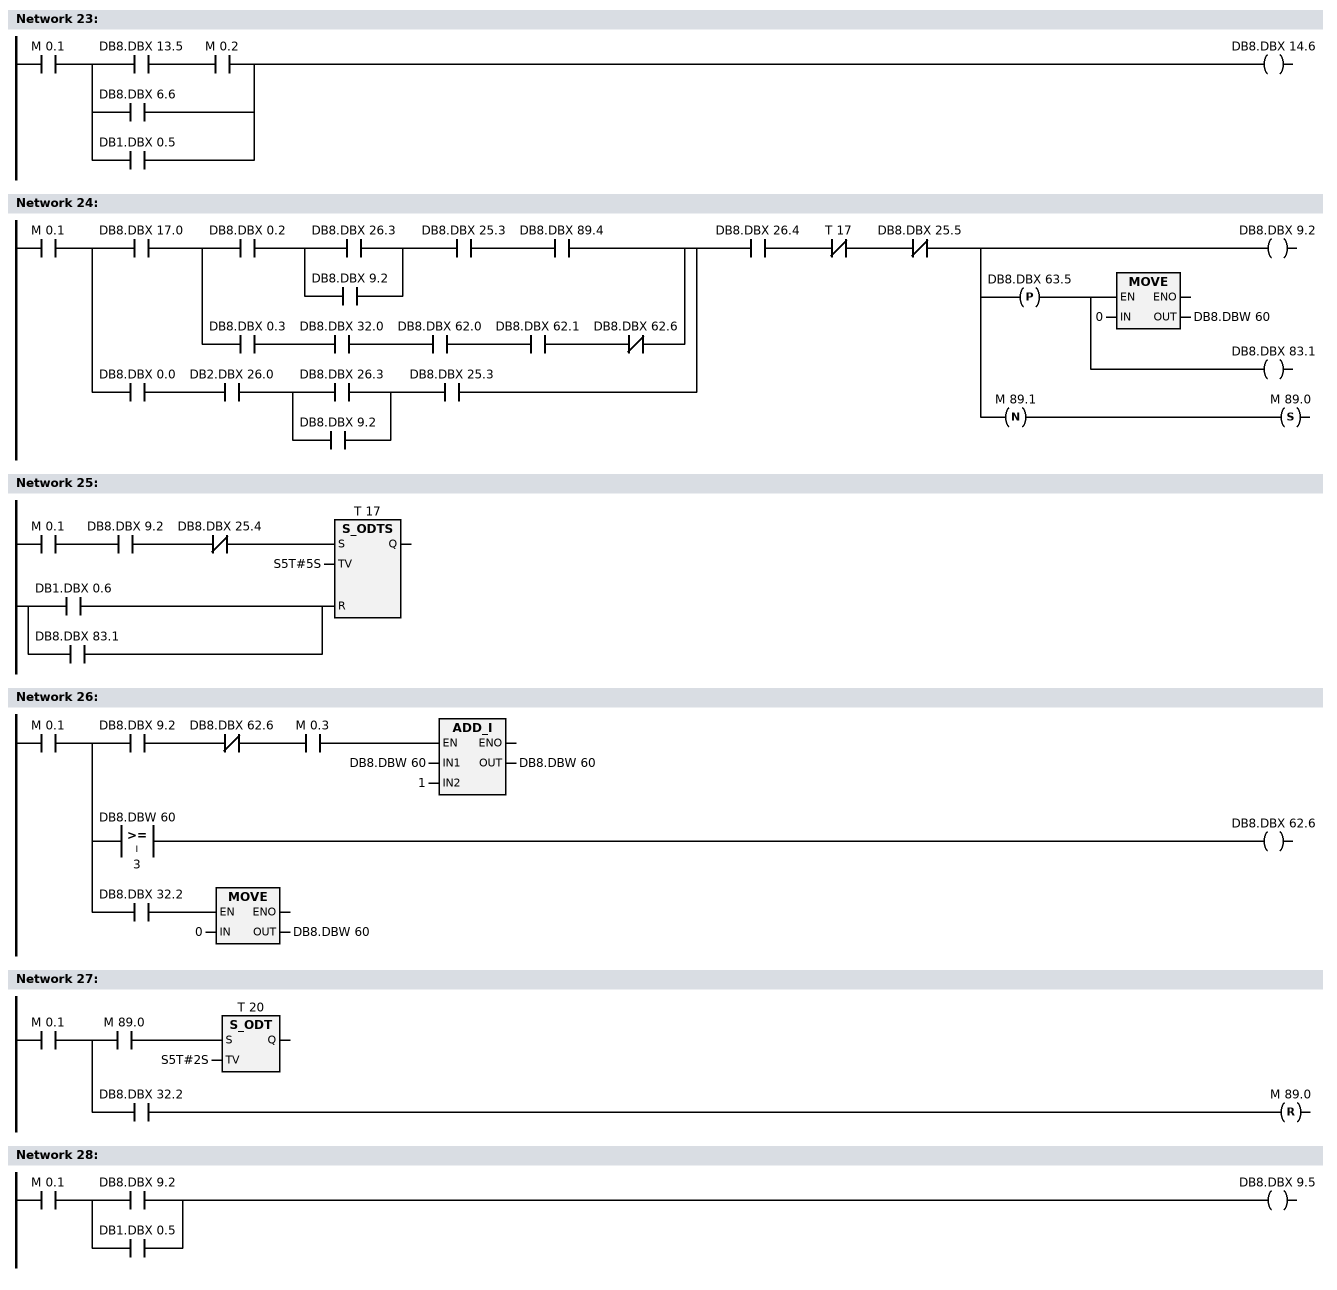
NETWORK
TITLE =
      A     M 0.1;
      A(;
      A     DB8.DBX 13.5;
      A     M 0.2;
      O     DB8.DBX 6.6;
      O     DB1.DBX 0.5;
      );
      =     DB8.DBX 14.6;
NETWORK
TITLE =
      A     M 0.1;
      A(;
      A     DB8.DBX 17.0;
      A(;
      A     DB8.DBX 0.2;
      A(;
      O     DB8.DBX 26.3;
      O     DB8.DBX 9.2;
      );
      A     DB8.DBX 25.3;
      A     DB8.DBX 89.4;
      O;
      A     DB8.DBX 0.3;
      A     DB8.DBX 32.0;
      A     DB8.DBX 62.0;
      A     DB8.DBX 62.1;
      AN    DB8.DBX 62.6;
      );
      O;
      A     DB8.DBX 0.0;
      A     DB2.DBX 26.0;
      A(;
      O     DB8.DBX 26.3;
      O     DB8.DBX 9.2;
      );
      A     DB8.DBX 25.3;
      );
      A     DB8.DBX 26.4;
      AN    T 17;
      AN    DB8.DBX 25.5;
      =     L 0.0;
      A     L 0.0;
      BLD   102;
      =     DB8.DBX 9.2;
      A     L 0.0;
      FP    DB8.DBX 63.5;
      =     L 0.1;
      A     L 0.1;
      JNB   M012;
      L     0;
      T     DB8.DBW 60;
M012: NOP   0;
      A     L 0.1;
      BLD   102;
      =     DB8.DBX 83.1;
      A     L 0.0;
      FN    M 89.1;
      S     M 89.0;
NETWORK
TITLE =
      A     M 0.1;
      A     DB8.DBX 9.2;
      AN    DB8.DBX 25.4;
      L     S5T#5S;
      SS    T 17;
      A(;
      O     DB1.DBX 0.6;
      O     DB8.DBX 83.1;
      );
      R     T 17;
      NOP   0;
      NOP   0;
      NOP   0;
NETWORK
TITLE =
      A     M 0.1;
      =     L 0.0;
      A     L 0.0;
      A     DB8.DBX 9.2;
      AN    DB8.DBX 62.6;
      A     M 0.3;
      JNB   M013;
      L     DB8.DBW 60;
      L     1;
      +I;
      T     DB8.DBW 60;
M013: NOP   0;
      A     L 0.0;
      A(;
      L     DB8.DBW 60;
      L     3;
      >=I;
      );
      =     DB8.DBX 62.6;
      A     L 0.0;
      A     DB8.DBX 32.2;
      JNB   M014;
      L     0;
      T     DB8.DBW 60;
M014: NOP   0;
NETWORK
TITLE =
      A     M 0.1;
      =     L 0.0;
      A     L 0.0;
      A     M 89.0;
      L     S5T#2S;
      SD    T 20;
      NOP   0;
      NOP   0;
      NOP   0;
      NOP   0;
      A     L 0.0;
      A     DB8.DBX 32.2;
      R     M 89.0;
NETWORK
TITLE =
      A     M 0.1;
      A(;
      O     DB8.DBX 9.2;
      O     DB1.DBX 0.5;
      );
      =     DB8.DBX 9.5;
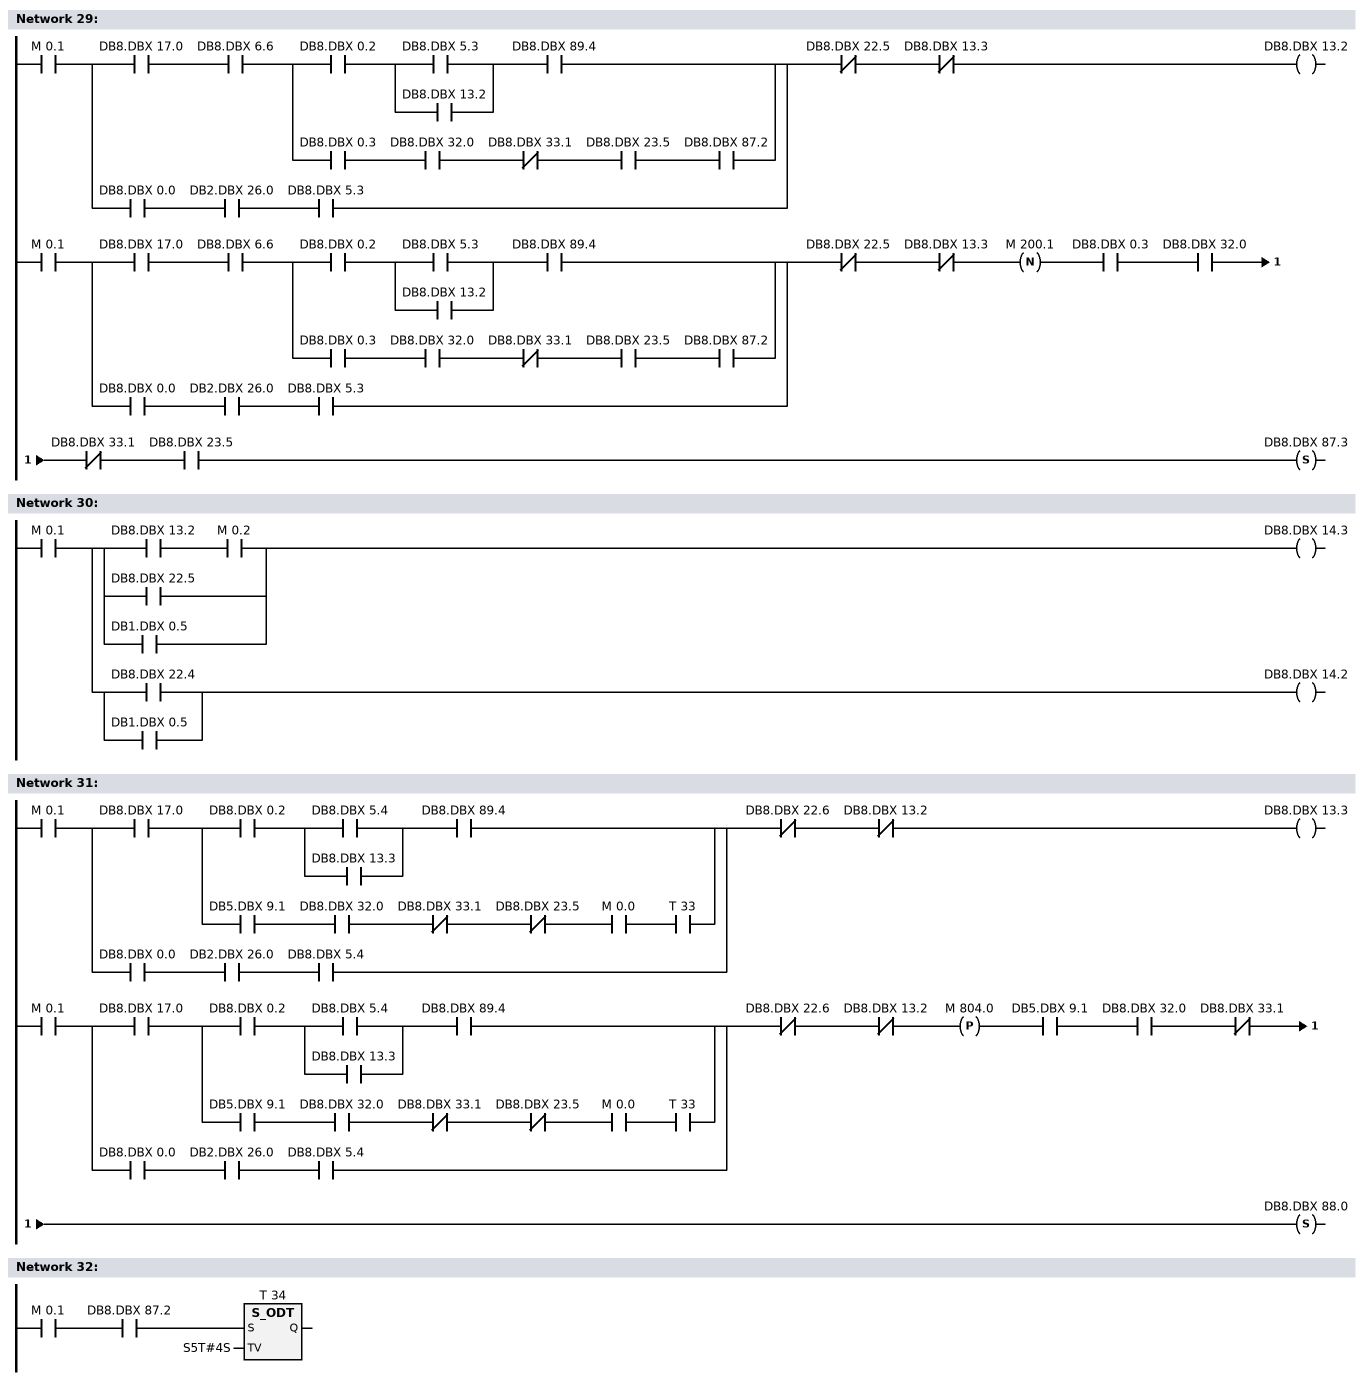
NETWORK
TITLE =
      A     M 0.1;
      A(;
      A     DB8.DBX 17.0;
      A     DB8.DBX 6.6;
      A(;
      A     DB8.DBX 0.2;
      A(;
      O     DB8.DBX 5.3;
      O     DB8.DBX 13.2;
      );
      A     DB8.DBX 89.4;
      O;
      A     DB8.DBX 0.3;
      A     DB8.DBX 32.0;
      AN    DB8.DBX 33.1;
      A     DB8.DBX 23.5;
      A     DB8.DBX 87.2;
      );
      O;
      A     DB8.DBX 0.0;
      A     DB2.DBX 26.0;
      A     DB8.DBX 5.3;
      );
      AN    DB8.DBX 22.5;
      AN    DB8.DBX 13.3;
      =     L 0.0;
      A     L 0.0;
      BLD   102;
      =     DB8.DBX 13.2;
      A(;
      A     L 0.0;
      FN    M 200.1;
      );
      A     DB8.DBX 0.3;
      A     DB8.DBX 32.0;
      AN    DB8.DBX 33.1;
      A     DB8.DBX 23.5;
      S     DB8.DBX 87.3;
NETWORK
TITLE =
      A     M 0.1;
      =     L 0.0;
      A     L 0.0;
      A(;
      A     DB8.DBX 13.2;
      A     M 0.2;
      O     DB8.DBX 22.5;
      O     DB1.DBX 0.5;
      );
      =     DB8.DBX 14.3;
      A     L 0.0;
      A(;
      O     DB8.DBX 22.4;
      O     DB1.DBX 0.5;
      );
      =     DB8.DBX 14.2;
NETWORK
TITLE =
      A     M 0.1;
      A(;
      A     DB8.DBX 17.0;
      A(;
      A     DB8.DBX 0.2;
      A(;
      O     DB8.DBX 5.4;
      O     DB8.DBX 13.3;
      );
      A     DB8.DBX 89.4;
      O;
      A     DB5.DBX 9.1;
      A     DB8.DBX 32.0;
      AN    DB8.DBX 33.1;
      AN    DB8.DBX 23.5;
      A     M 0.0;
      A     T 33;
      );
      O;
      A     DB8.DBX 0.0;
      A     DB2.DBX 26.0;
      A     DB8.DBX 5.4;
      );
      AN    DB8.DBX 22.6;
      AN    DB8.DBX 13.2;
      =     L 0.0;
      A     L 0.0;
      BLD   102;
      =     DB8.DBX 13.3;
      A(;
      A     L 0.0;
      FP    M 804.0;
      );
      A     DB5.DBX 9.1;
      A     DB8.DBX 32.0;
      AN    DB8.DBX 33.1;
      S     DB8.DBX 88.0;
NETWORK
TITLE =
      A     M 0.1;
      A     DB8.DBX 87.2;
      L     S5T#4S;
      SD    T 34;
      NOP   0;
      NOP   0;
      NOP   0;
      NOP   0;
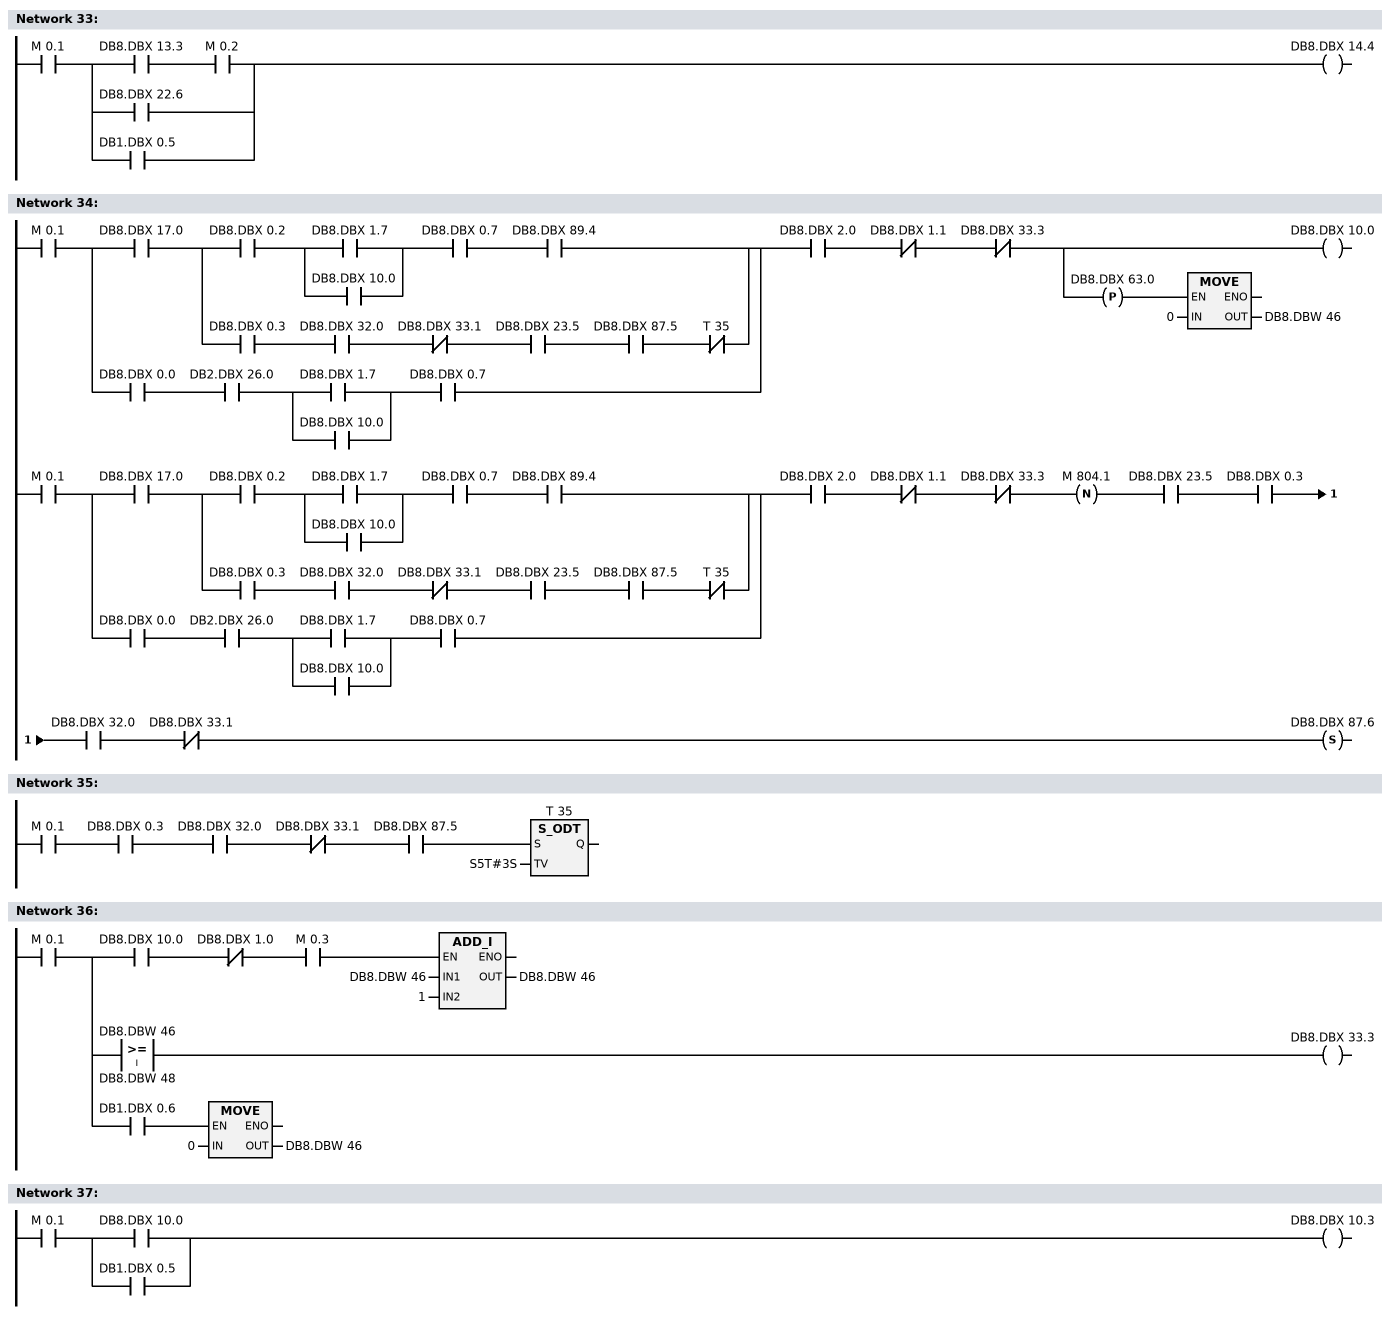
NETWORK
TITLE =
      A     M 0.1;
      A(;
      A     DB8.DBX 13.3;
      A     M 0.2;
      O     DB8.DBX 22.6;
      O     DB1.DBX 0.5;
      );
      =     DB8.DBX 14.4;
NETWORK
TITLE =
      A     M 0.1;
      A(;
      A     DB8.DBX 17.0;
      A(;
      A     DB8.DBX 0.2;
      A(;
      O     DB8.DBX 1.7;
      O     DB8.DBX 10.0;
      );
      A     DB8.DBX 0.7;
      A     DB8.DBX 89.4;
      O;
      A     DB8.DBX 0.3;
      A     DB8.DBX 32.0;
      AN    DB8.DBX 33.1;
      A     DB8.DBX 23.5;
      A     DB8.DBX 87.5;
      AN    T 35;
      );
      O;
      A     DB8.DBX 0.0;
      A     DB2.DBX 26.0;
      A(;
      O     DB8.DBX 1.7;
      O     DB8.DBX 10.0;
      );
      A     DB8.DBX 0.7;
      );
      A     DB8.DBX 2.0;
      AN    DB8.DBX 1.1;
      AN    DB8.DBX 33.3;
      =     L 0.0;
      A     L 0.0;
      BLD   102;
      =     DB8.DBX 10.0;
      A     L 0.0;
      FP    DB8.DBX 63.0;
      JNB   M015;
      L     0;
      T     DB8.DBW 46;
M015: NOP   0;
      A(;
      A     L 0.0;
      FN    M 804.1;
      );
      A     DB8.DBX 23.5;
      A     DB8.DBX 0.3;
      A     DB8.DBX 32.0;
      AN    DB8.DBX 33.1;
      S     DB8.DBX 87.6;
NETWORK
TITLE =
      A     M 0.1;
      A     DB8.DBX 0.3;
      A     DB8.DBX 32.0;
      AN    DB8.DBX 33.1;
      A     DB8.DBX 87.5;
      L     S5T#3S;
      SD    T 35;
      NOP   0;
      NOP   0;
      NOP   0;
      NOP   0;
NETWORK
TITLE =
      A     M 0.1;
      =     L 0.0;
      A     L 0.0;
      A     DB8.DBX 10.0;
      AN    DB8.DBX 1.0;
      A     M 0.3;
      JNB   M016;
      L     DB8.DBW 46;
      L     1;
      +I;
      T     DB8.DBW 46;
M016: NOP   0;
      A     L 0.0;
      A(;
      L     DB8.DBW 46;
      L     DB8.DBW 48;
      >=I;
      );
      =     DB8.DBX 33.3;
      A     L 0.0;
      A     DB1.DBX 0.6;
      JNB   M017;
      L     0;
      T     DB8.DBW 46;
M017: NOP   0;
NETWORK
TITLE =
      A     M 0.1;
      A(;
      O     DB8.DBX 10.0;
      O     DB1.DBX 0.5;
      );
      =     DB8.DBX 10.3;
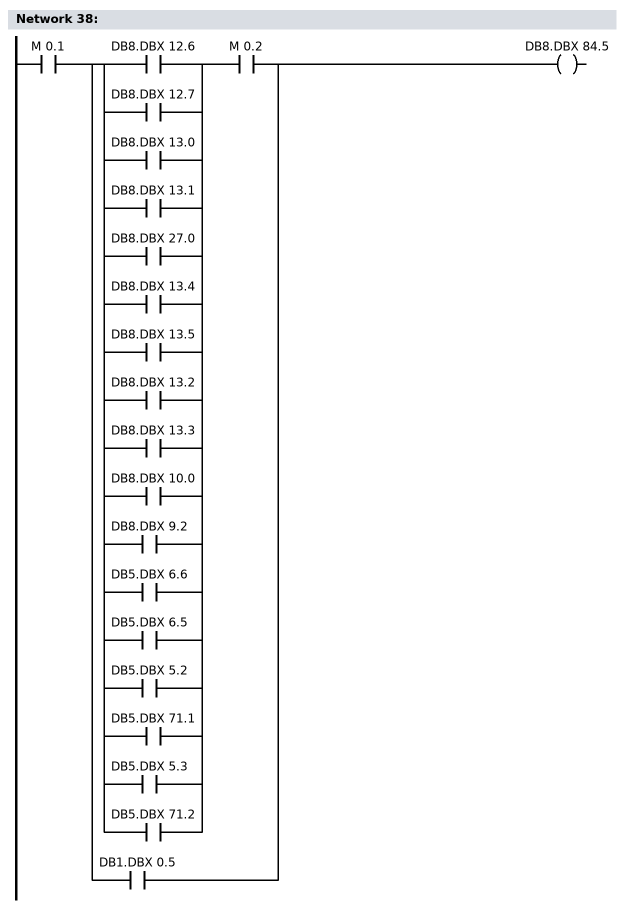
NETWORK
TITLE =
      A     M 0.1;
      A(;
      A(;
      O     DB8.DBX 12.6;
      O     DB8.DBX 12.7;
      O     DB8.DBX 13.0;
      O     DB8.DBX 13.1;
      O     DB8.DBX 27.0;
      O     DB8.DBX 13.4;
      O     DB8.DBX 13.5;
      O     DB8.DBX 13.2;
      O     DB8.DBX 13.3;
      O     DB8.DBX 10.0;
      O     DB8.DBX 9.2;
      O     DB5.DBX 6.6;
      O     DB5.DBX 6.5;
      O     DB5.DBX 5.2;
      O     DB5.DBX 71.1;
      O     DB5.DBX 5.3;
      O     DB5.DBX 71.2;
      );
      A     M 0.2;
      O     DB1.DBX 0.5;
      );
      =     DB8.DBX 84.5;
END_FUNCTION

FUNCTION FC 14 : VOID
AUTHOR : Arun
VERSION : 0.1
BEGIN
// (block stored without names or comments; labels and parameter names are numbered)
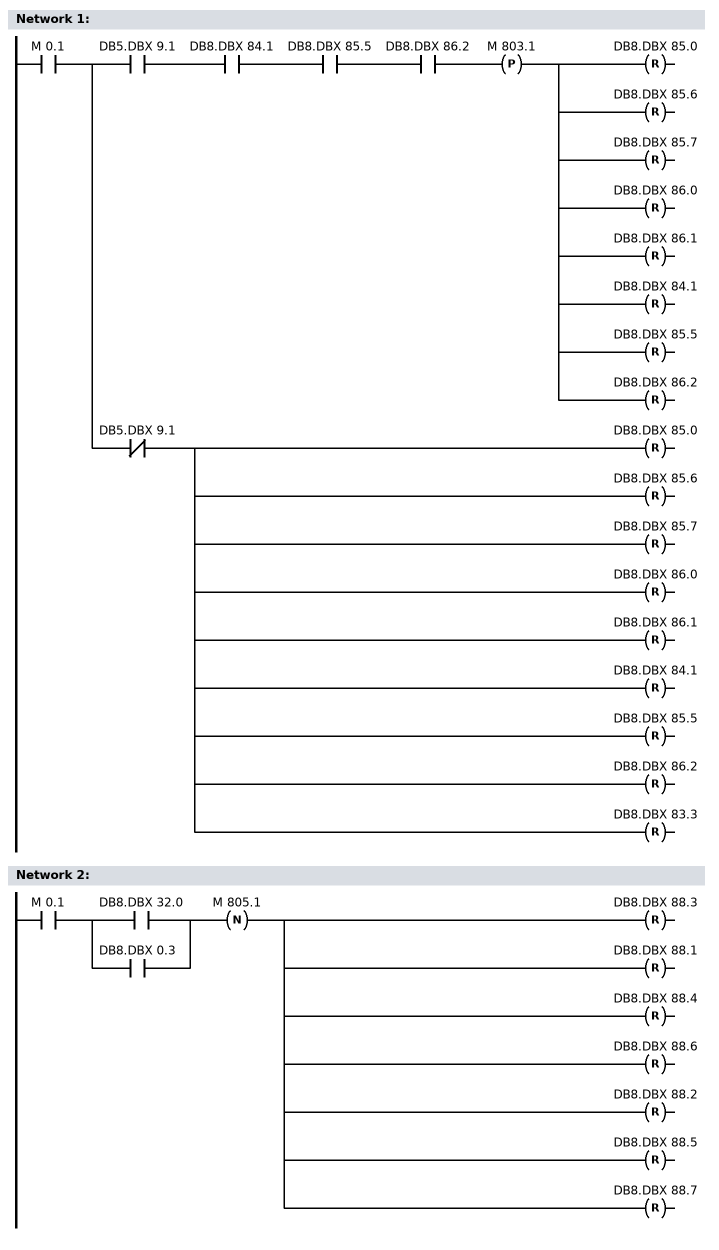
NETWORK
TITLE =
      A     M 0.1;
      =     L 0.0;
      A     L 0.0;
      A     DB5.DBX 9.1;
      A     DB8.DBX 84.1;
      A     DB8.DBX 85.5;
      A     DB8.DBX 86.2;
      FP    M 803.1;
      R     DB8.DBX 85.0;
      R     DB8.DBX 85.6;
      R     DB8.DBX 85.7;
      R     DB8.DBX 86.0;
      R     DB8.DBX 86.1;
      R     DB8.DBX 84.1;
      R     DB8.DBX 85.5;
      R     DB8.DBX 86.2;
      A     L 0.0;
      AN    DB5.DBX 9.1;
      R     DB8.DBX 85.0;
      R     DB8.DBX 85.6;
      R     DB8.DBX 85.7;
      R     DB8.DBX 86.0;
      R     DB8.DBX 86.1;
      R     DB8.DBX 84.1;
      R     DB8.DBX 85.5;
      R     DB8.DBX 86.2;
      R     DB8.DBX 83.3;
NETWORK
TITLE =
      A     M 0.1;
      A(;
      O     DB8.DBX 32.0;
      O     DB8.DBX 0.3;
      );
      FN    M 805.1;
      R     DB8.DBX 88.3;
      R     DB8.DBX 88.1;
      R     DB8.DBX 88.4;
      R     DB8.DBX 88.6;
      R     DB8.DBX 88.2;
      R     DB8.DBX 88.5;
      R     DB8.DBX 88.7;
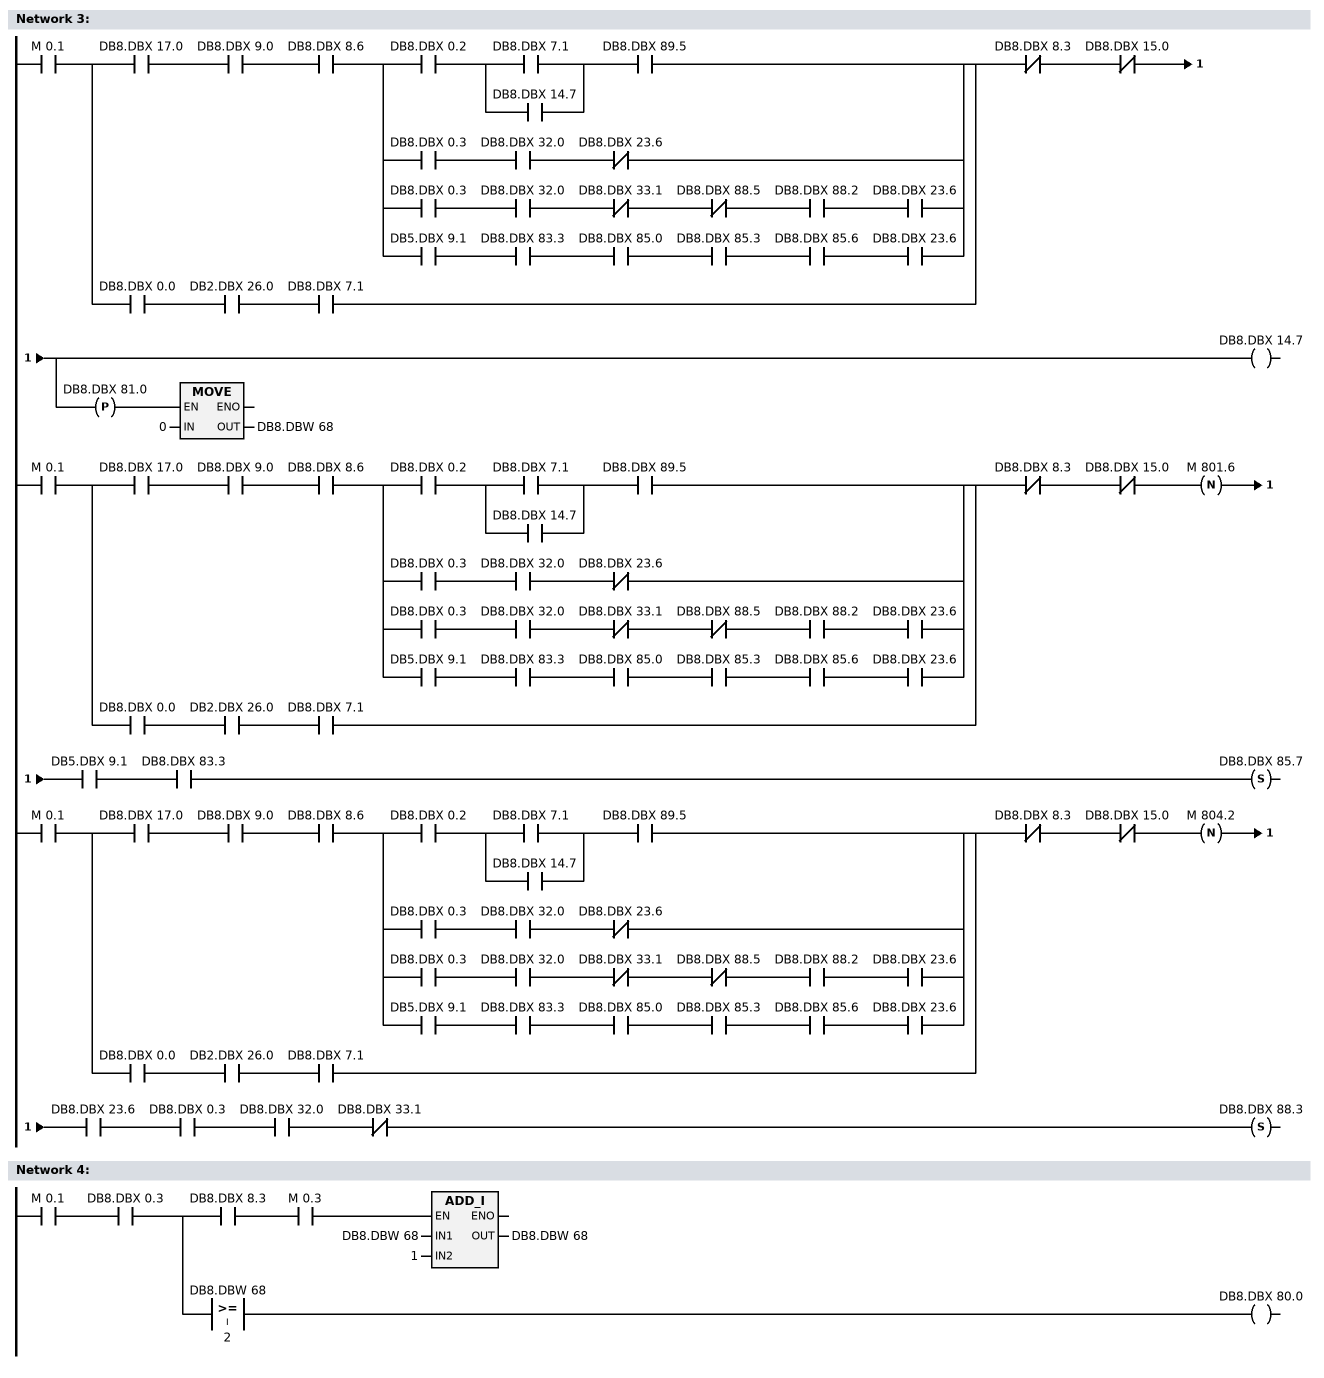
NETWORK
TITLE =
      A     M 0.1;
      A(;
      A     DB8.DBX 17.0;
      A     DB8.DBX 9.0;
      A     DB8.DBX 8.6;
      A(;
      A     DB8.DBX 0.2;
      A(;
      O     DB8.DBX 7.1;
      O     DB8.DBX 14.7;
      );
      A     DB8.DBX 89.5;
      O;
      A     DB8.DBX 0.3;
      A     DB8.DBX 32.0;
      AN    DB8.DBX 23.6;
      O;
      A     DB8.DBX 0.3;
      A     DB8.DBX 32.0;
      AN    DB8.DBX 33.1;
      AN    DB8.DBX 88.5;
      A     DB8.DBX 88.2;
      A     DB8.DBX 23.6;
      O;
      A     DB5.DBX 9.1;
      A     DB8.DBX 83.3;
      A     DB8.DBX 85.0;
      A     DB8.DBX 85.3;
      A     DB8.DBX 85.6;
      A     DB8.DBX 23.6;
      );
      O;
      A     DB8.DBX 0.0;
      A     DB2.DBX 26.0;
      A     DB8.DBX 7.1;
      );
      AN    DB8.DBX 8.3;
      AN    DB8.DBX 15.0;
      =     L 0.0;
      A     L 0.0;
      BLD   102;
      =     DB8.DBX 14.7;
      A     L 0.0;
      FP    DB8.DBX 81.0;
      JNB   M001;
      L     0;
      T     DB8.DBW 68;
M001: NOP   0;
      A(;
      A     L 0.0;
      FN    M 801.6;
      );
      A     DB5.DBX 9.1;
      A     DB8.DBX 83.3;
      S     DB8.DBX 85.7;
      A(;
      A     L 0.0;
      FN    M 804.2;
      );
      A     DB8.DBX 23.6;
      A     DB8.DBX 0.3;
      A     DB8.DBX 32.0;
      AN    DB8.DBX 33.1;
      S     DB8.DBX 88.3;
NETWORK
TITLE =
      A     M 0.1;
      A     DB8.DBX 0.3;
      =     L 0.0;
      A     L 0.0;
      A     DB8.DBX 8.3;
      A     M 0.3;
      JNB   M002;
      L     DB8.DBW 68;
      L     1;
      +I;
      T     DB8.DBW 68;
M002: NOP   0;
      A     L 0.0;
      A(;
      L     DB8.DBW 68;
      L     2;
      >=I;
      );
      =     DB8.DBX 80.0;
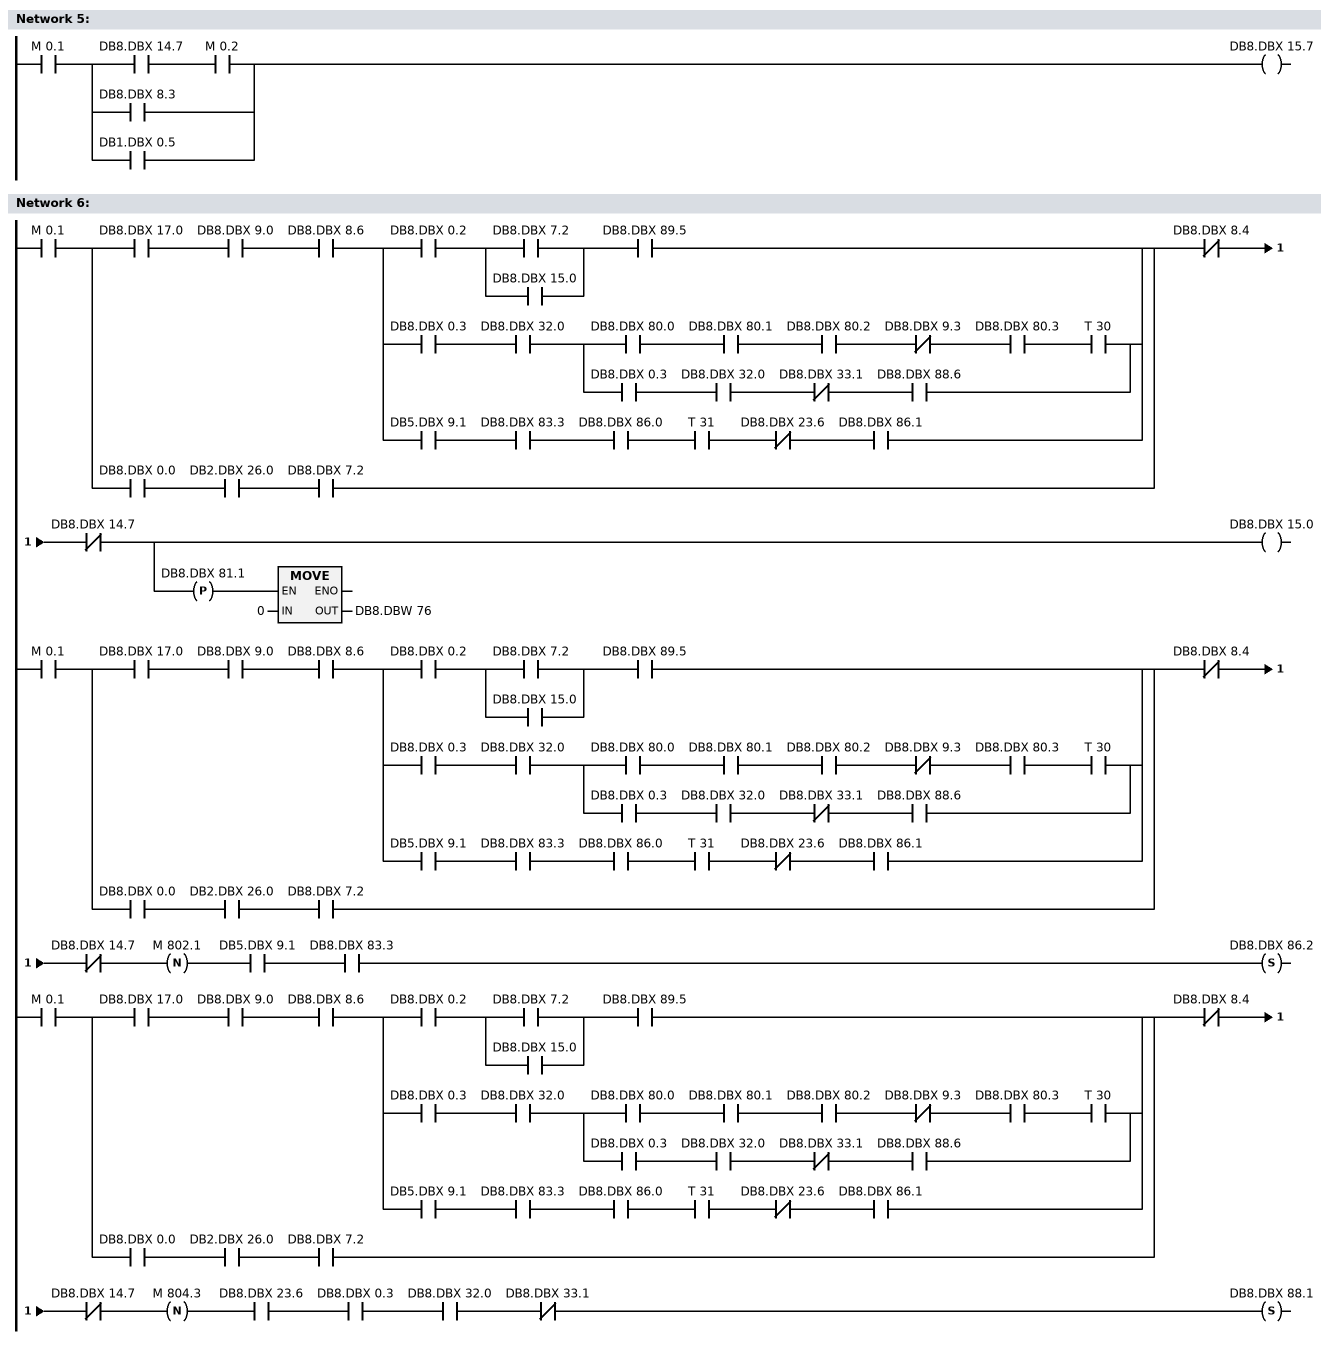
NETWORK
TITLE =
      A     M 0.1;
      A(;
      A     DB8.DBX 14.7;
      A     M 0.2;
      O     DB8.DBX 8.3;
      O     DB1.DBX 0.5;
      );
      =     DB8.DBX 15.7;
NETWORK
TITLE =
      A     M 0.1;
      A(;
      A     DB8.DBX 17.0;
      A     DB8.DBX 9.0;
      A     DB8.DBX 8.6;
      A(;
      A     DB8.DBX 0.2;
      A(;
      O     DB8.DBX 7.2;
      O     DB8.DBX 15.0;
      );
      A     DB8.DBX 89.5;
      O;
      A     DB8.DBX 0.3;
      A     DB8.DBX 32.0;
      A(;
      A     DB8.DBX 80.0;
      A     DB8.DBX 80.1;
      A     DB8.DBX 80.2;
      AN    DB8.DBX 9.3;
      A     DB8.DBX 80.3;
      A     T 30;
      O;
      A     DB8.DBX 0.3;
      A     DB8.DBX 32.0;
      AN    DB8.DBX 33.1;
      A     DB8.DBX 88.6;
      );
      O;
      A     DB5.DBX 9.1;
      A     DB8.DBX 83.3;
      A     DB8.DBX 86.0;
      A     T 31;
      AN    DB8.DBX 23.6;
      A     DB8.DBX 86.1;
      );
      O;
      A     DB8.DBX 0.0;
      A     DB2.DBX 26.0;
      A     DB8.DBX 7.2;
      );
      AN    DB8.DBX 8.4;
      AN    DB8.DBX 14.7;
      =     L 0.0;
      A     L 0.0;
      BLD   102;
      =     DB8.DBX 15.0;
      A     L 0.0;
      FP    DB8.DBX 81.1;
      JNB   M003;
      L     0;
      T     DB8.DBW 76;
M003: NOP   0;
      A(;
      A     L 0.0;
      FN    M 802.1;
      );
      A     DB5.DBX 9.1;
      A     DB8.DBX 83.3;
      S     DB8.DBX 86.2;
      A(;
      A     L 0.0;
      FN    M 804.3;
      );
      A     DB8.DBX 23.6;
      A     DB8.DBX 0.3;
      A     DB8.DBX 32.0;
      AN    DB8.DBX 33.1;
      S     DB8.DBX 88.1;
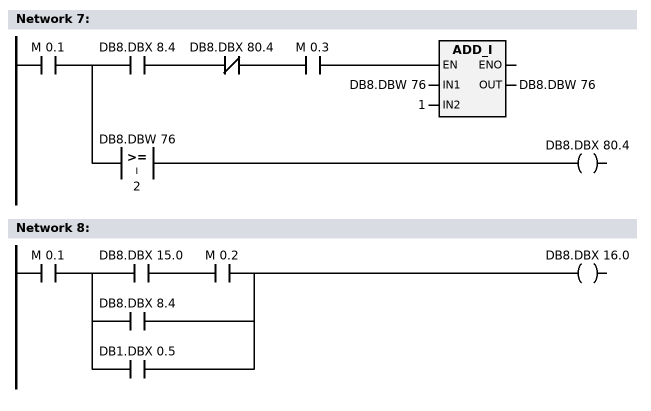
NETWORK
TITLE =
      A     M 0.1;
      =     L 0.0;
      A     L 0.0;
      A     DB8.DBX 8.4;
      AN    DB8.DBX 80.4;
      A     M 0.3;
      JNB   M004;
      L     DB8.DBW 76;
      L     1;
      +I;
      T     DB8.DBW 76;
M004: NOP   0;
      A     L 0.0;
      A(;
      L     DB8.DBW 76;
      L     2;
      >=I;
      );
      =     DB8.DBX 80.4;
NETWORK
TITLE =
      A     M 0.1;
      A(;
      A     DB8.DBX 15.0;
      A     M 0.2;
      O     DB8.DBX 8.4;
      O     DB1.DBX 0.5;
      );
      =     DB8.DBX 16.0;
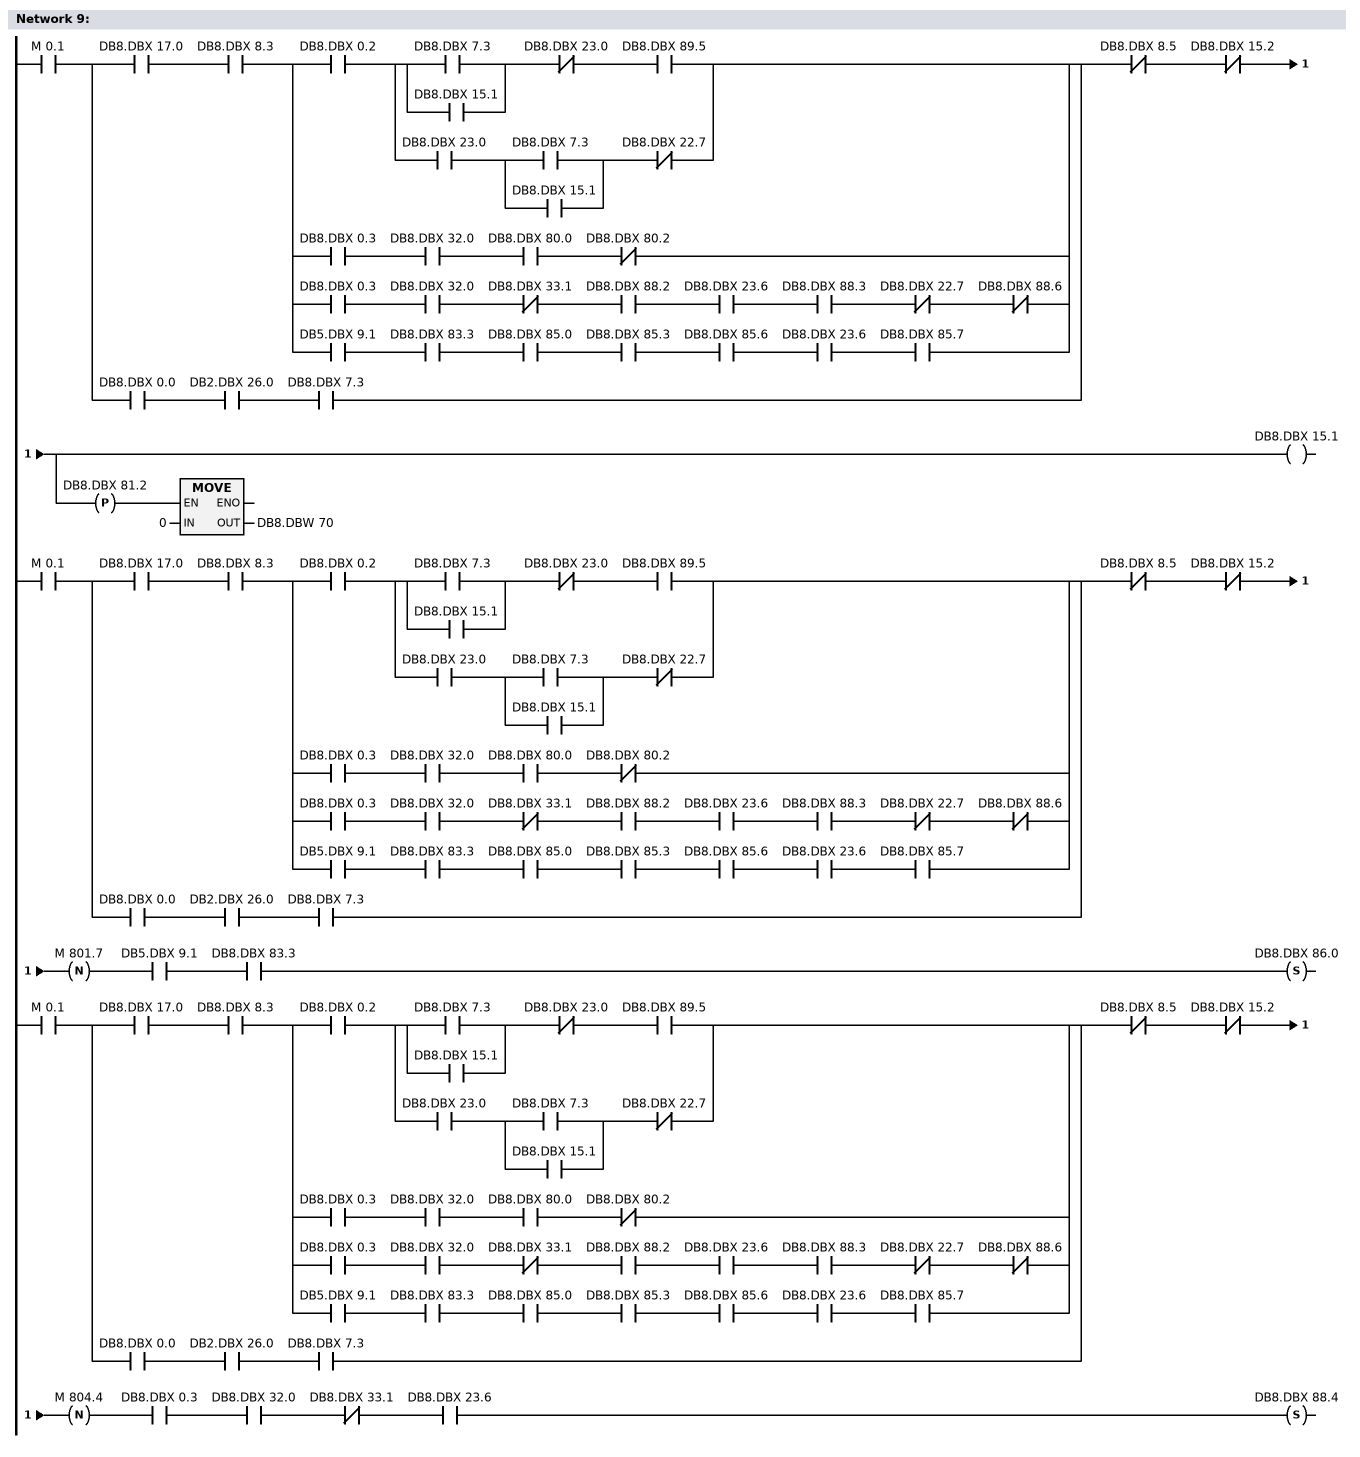
NETWORK
TITLE =
      A     M 0.1;
      A(;
      A     DB8.DBX 17.0;
      A     DB8.DBX 8.3;
      A(;
      A     DB8.DBX 0.2;
      A(;
      A(;
      O     DB8.DBX 7.3;
      O     DB8.DBX 15.1;
      );
      AN    DB8.DBX 23.0;
      A     DB8.DBX 89.5;
      O;
      A     DB8.DBX 23.0;
      A(;
      O     DB8.DBX 7.3;
      O     DB8.DBX 15.1;
      );
      AN    DB8.DBX 22.7;
      );
      O;
      A     DB8.DBX 0.3;
      A     DB8.DBX 32.0;
      A     DB8.DBX 80.0;
      AN    DB8.DBX 80.2;
      O;
      A     DB8.DBX 0.3;
      A     DB8.DBX 32.0;
      AN    DB8.DBX 33.1;
      A     DB8.DBX 88.2;
      A     DB8.DBX 23.6;
      A     DB8.DBX 88.3;
      AN    DB8.DBX 22.7;
      AN    DB8.DBX 88.6;
      O;
      A     DB5.DBX 9.1;
      A     DB8.DBX 83.3;
      A     DB8.DBX 85.0;
      A     DB8.DBX 85.3;
      A     DB8.DBX 85.6;
      A     DB8.DBX 23.6;
      A     DB8.DBX 85.7;
      );
      O;
      A     DB8.DBX 0.0;
      A     DB2.DBX 26.0;
      A     DB8.DBX 7.3;
      );
      AN    DB8.DBX 8.5;
      AN    DB8.DBX 15.2;
      =     L 0.0;
      A     L 0.0;
      BLD   102;
      =     DB8.DBX 15.1;
      A     L 0.0;
      FP    DB8.DBX 81.2;
      JNB   M005;
      L     0;
      T     DB8.DBW 70;
M005: NOP   0;
      A(;
      A     L 0.0;
      FN    M 801.7;
      );
      A     DB5.DBX 9.1;
      A     DB8.DBX 83.3;
      S     DB8.DBX 86.0;
      A(;
      A     L 0.0;
      FN    M 804.4;
      );
      A     DB8.DBX 0.3;
      A     DB8.DBX 32.0;
      AN    DB8.DBX 33.1;
      A     DB8.DBX 23.6;
      S     DB8.DBX 88.4;
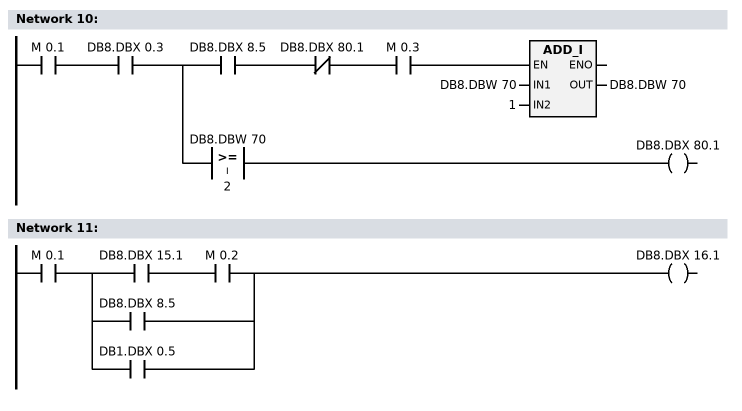
NETWORK
TITLE =
      A     M 0.1;
      A     DB8.DBX 0.3;
      =     L 0.0;
      A     L 0.0;
      A     DB8.DBX 8.5;
      AN    DB8.DBX 80.1;
      A     M 0.3;
      JNB   M006;
      L     DB8.DBW 70;
      L     1;
      +I;
      T     DB8.DBW 70;
M006: NOP   0;
      A     L 0.0;
      A(;
      L     DB8.DBW 70;
      L     2;
      >=I;
      );
      =     DB8.DBX 80.1;
NETWORK
TITLE =
      A     M 0.1;
      A(;
      A     DB8.DBX 15.1;
      A     M 0.2;
      O     DB8.DBX 8.5;
      O     DB1.DBX 0.5;
      );
      =     DB8.DBX 16.1;
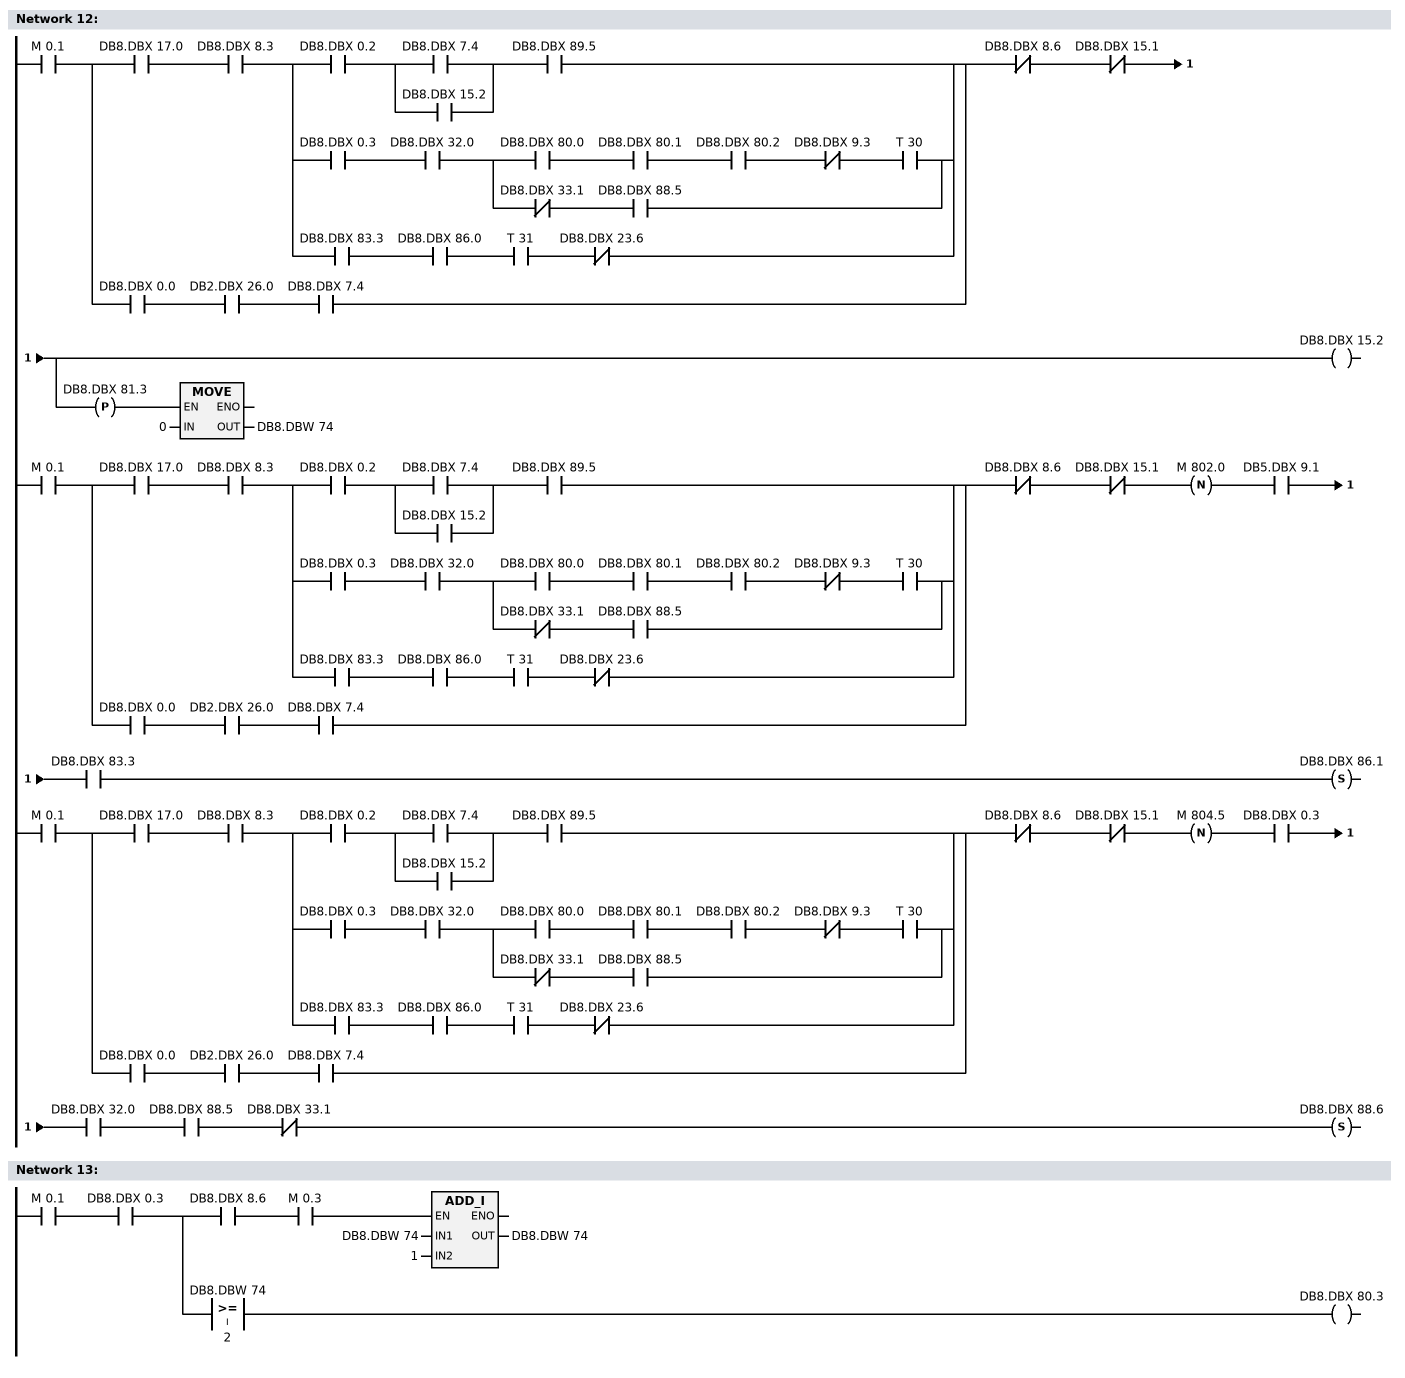
NETWORK
TITLE =
      A     M 0.1;
      A(;
      A     DB8.DBX 17.0;
      A     DB8.DBX 8.3;
      A(;
      A     DB8.DBX 0.2;
      A(;
      O     DB8.DBX 7.4;
      O     DB8.DBX 15.2;
      );
      A     DB8.DBX 89.5;
      O;
      A     DB8.DBX 0.3;
      A     DB8.DBX 32.0;
      A(;
      A     DB8.DBX 80.0;
      A     DB8.DBX 80.1;
      A     DB8.DBX 80.2;
      AN    DB8.DBX 9.3;
      A     T 30;
      O;
      AN    DB8.DBX 33.1;
      A     DB8.DBX 88.5;
      );
      O;
      A     DB8.DBX 83.3;
      A     DB8.DBX 86.0;
      A     T 31;
      AN    DB8.DBX 23.6;
      );
      O;
      A     DB8.DBX 0.0;
      A     DB2.DBX 26.0;
      A     DB8.DBX 7.4;
      );
      AN    DB8.DBX 8.6;
      AN    DB8.DBX 15.1;
      =     L 0.0;
      A     L 0.0;
      BLD   102;
      =     DB8.DBX 15.2;
      A     L 0.0;
      FP    DB8.DBX 81.3;
      JNB   M007;
      L     0;
      T     DB8.DBW 74;
M007: NOP   0;
      A(;
      A     L 0.0;
      FN    M 802.0;
      );
      A     DB5.DBX 9.1;
      A     DB8.DBX 83.3;
      S     DB8.DBX 86.1;
      A(;
      A     L 0.0;
      FN    M 804.5;
      );
      A     DB8.DBX 0.3;
      A     DB8.DBX 32.0;
      A     DB8.DBX 88.5;
      AN    DB8.DBX 33.1;
      S     DB8.DBX 88.6;
NETWORK
TITLE =
      A     M 0.1;
      A     DB8.DBX 0.3;
      =     L 0.0;
      A     L 0.0;
      A     DB8.DBX 8.6;
      A     M 0.3;
      JNB   M008;
      L     DB8.DBW 74;
      L     1;
      +I;
      T     DB8.DBW 74;
M008: NOP   0;
      A     L 0.0;
      A(;
      L     DB8.DBW 74;
      L     2;
      >=I;
      );
      =     DB8.DBX 80.3;
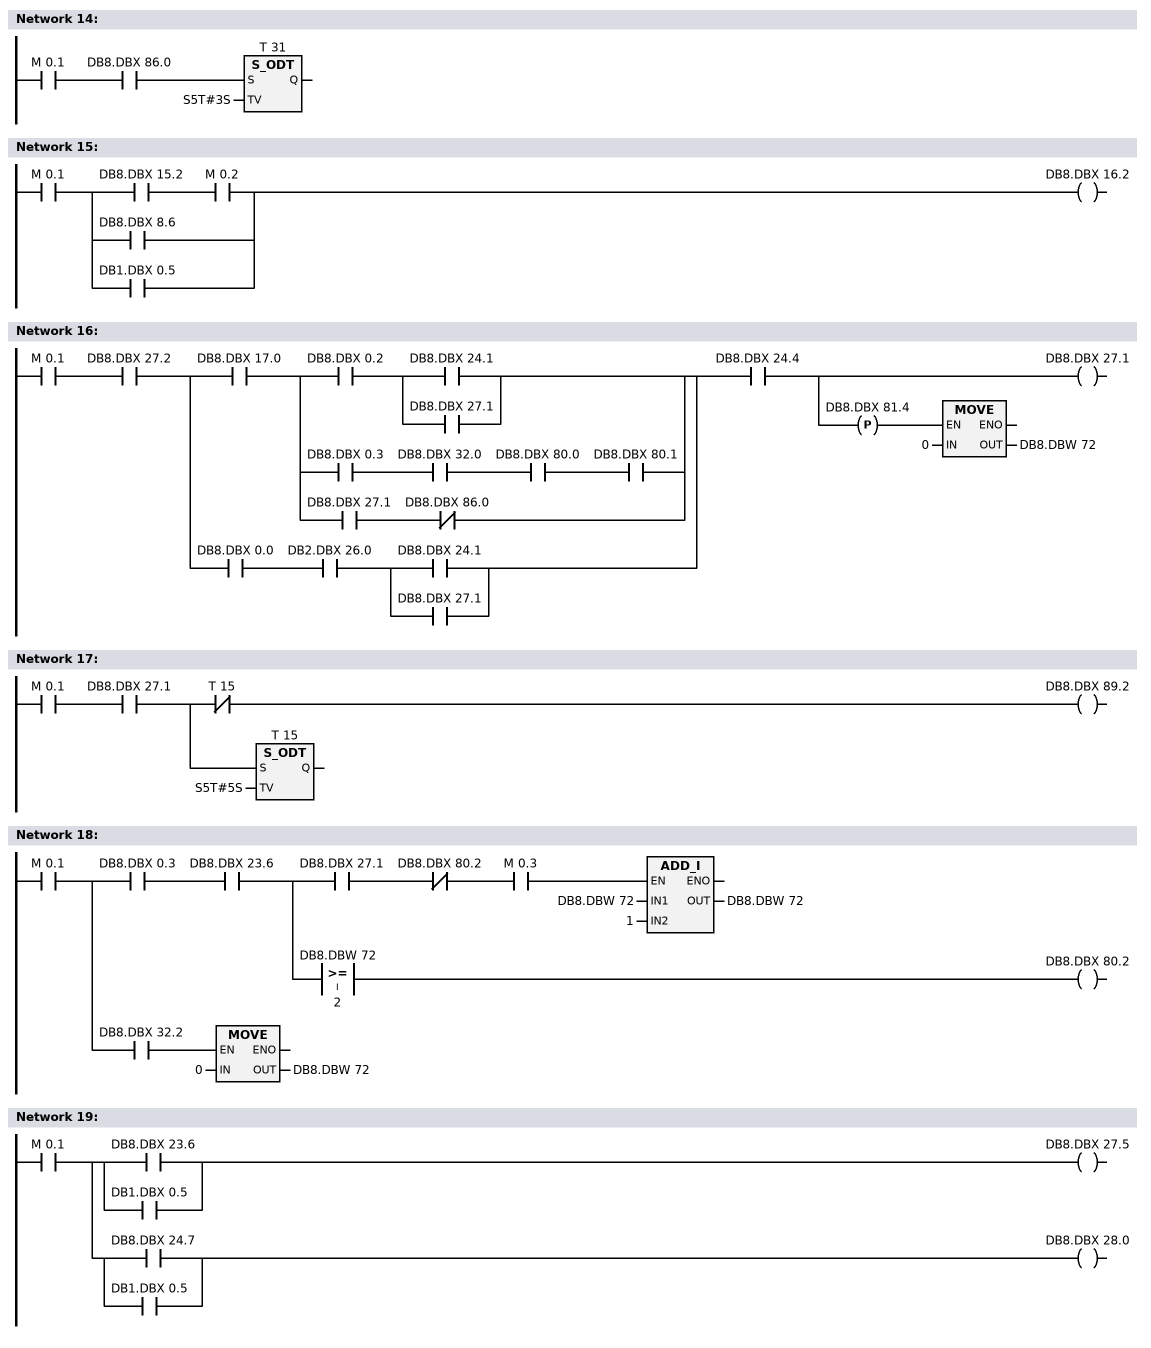
NETWORK
TITLE =
      A     M 0.1;
      A     DB8.DBX 86.0;
      L     S5T#3S;
      SD    T 31;
      NOP   0;
      NOP   0;
      NOP   0;
      NOP   0;
NETWORK
TITLE =
      A     M 0.1;
      A(;
      A     DB8.DBX 15.2;
      A     M 0.2;
      O     DB8.DBX 8.6;
      O     DB1.DBX 0.5;
      );
      =     DB8.DBX 16.2;
NETWORK
TITLE =
      A     M 0.1;
      A     DB8.DBX 27.2;
      A(;
      A     DB8.DBX 17.0;
      A(;
      A     DB8.DBX 0.2;
      A(;
      O     DB8.DBX 24.1;
      O     DB8.DBX 27.1;
      );
      O;
      A     DB8.DBX 0.3;
      A     DB8.DBX 32.0;
      A     DB8.DBX 80.0;
      A     DB8.DBX 80.1;
      O;
      A     DB8.DBX 27.1;
      AN    DB8.DBX 86.0;
      );
      O;
      A     DB8.DBX 0.0;
      A     DB2.DBX 26.0;
      A(;
      O     DB8.DBX 24.1;
      O     DB8.DBX 27.1;
      );
      );
      A     DB8.DBX 24.4;
      =     L 0.0;
      A     L 0.0;
      BLD   102;
      =     DB8.DBX 27.1;
      A     L 0.0;
      FP    DB8.DBX 81.4;
      JNB   M009;
      L     0;
      T     DB8.DBW 72;
M009: NOP   0;
NETWORK
TITLE =
      A     M 0.1;
      A     DB8.DBX 27.1;
      =     L 0.0;
      A     L 0.0;
      AN    T 15;
      =     DB8.DBX 89.2;
      A     L 0.0;
      L     S5T#5S;
      SD    T 15;
      NOP   0;
      NOP   0;
      NOP   0;
      NOP   0;
NETWORK
TITLE =
      A     M 0.1;
      =     L 0.0;
      A     L 0.0;
      A     DB8.DBX 0.3;
      A     DB8.DBX 23.6;
      =     L 0.1;
      A     L 0.1;
      A     DB8.DBX 27.1;
      AN    DB8.DBX 80.2;
      A     M 0.3;
      JNB   M010;
      L     DB8.DBW 72;
      L     1;
      +I;
      T     DB8.DBW 72;
M010: NOP   0;
      A     L 0.1;
      A(;
      L     DB8.DBW 72;
      L     2;
      >=I;
      );
      =     DB8.DBX 80.2;
      A     L 0.0;
      A     DB8.DBX 32.2;
      JNB   M011;
      L     0;
      T     DB8.DBW 72;
M011: NOP   0;
NETWORK
TITLE =
      A     M 0.1;
      =     L 0.0;
      A     L 0.0;
      A(;
      O     DB8.DBX 23.6;
      O     DB1.DBX 0.5;
      );
      =     DB8.DBX 27.5;
      A     L 0.0;
      A(;
      O     DB8.DBX 24.7;
      O     DB1.DBX 0.5;
      );
      =     DB8.DBX 28.0;
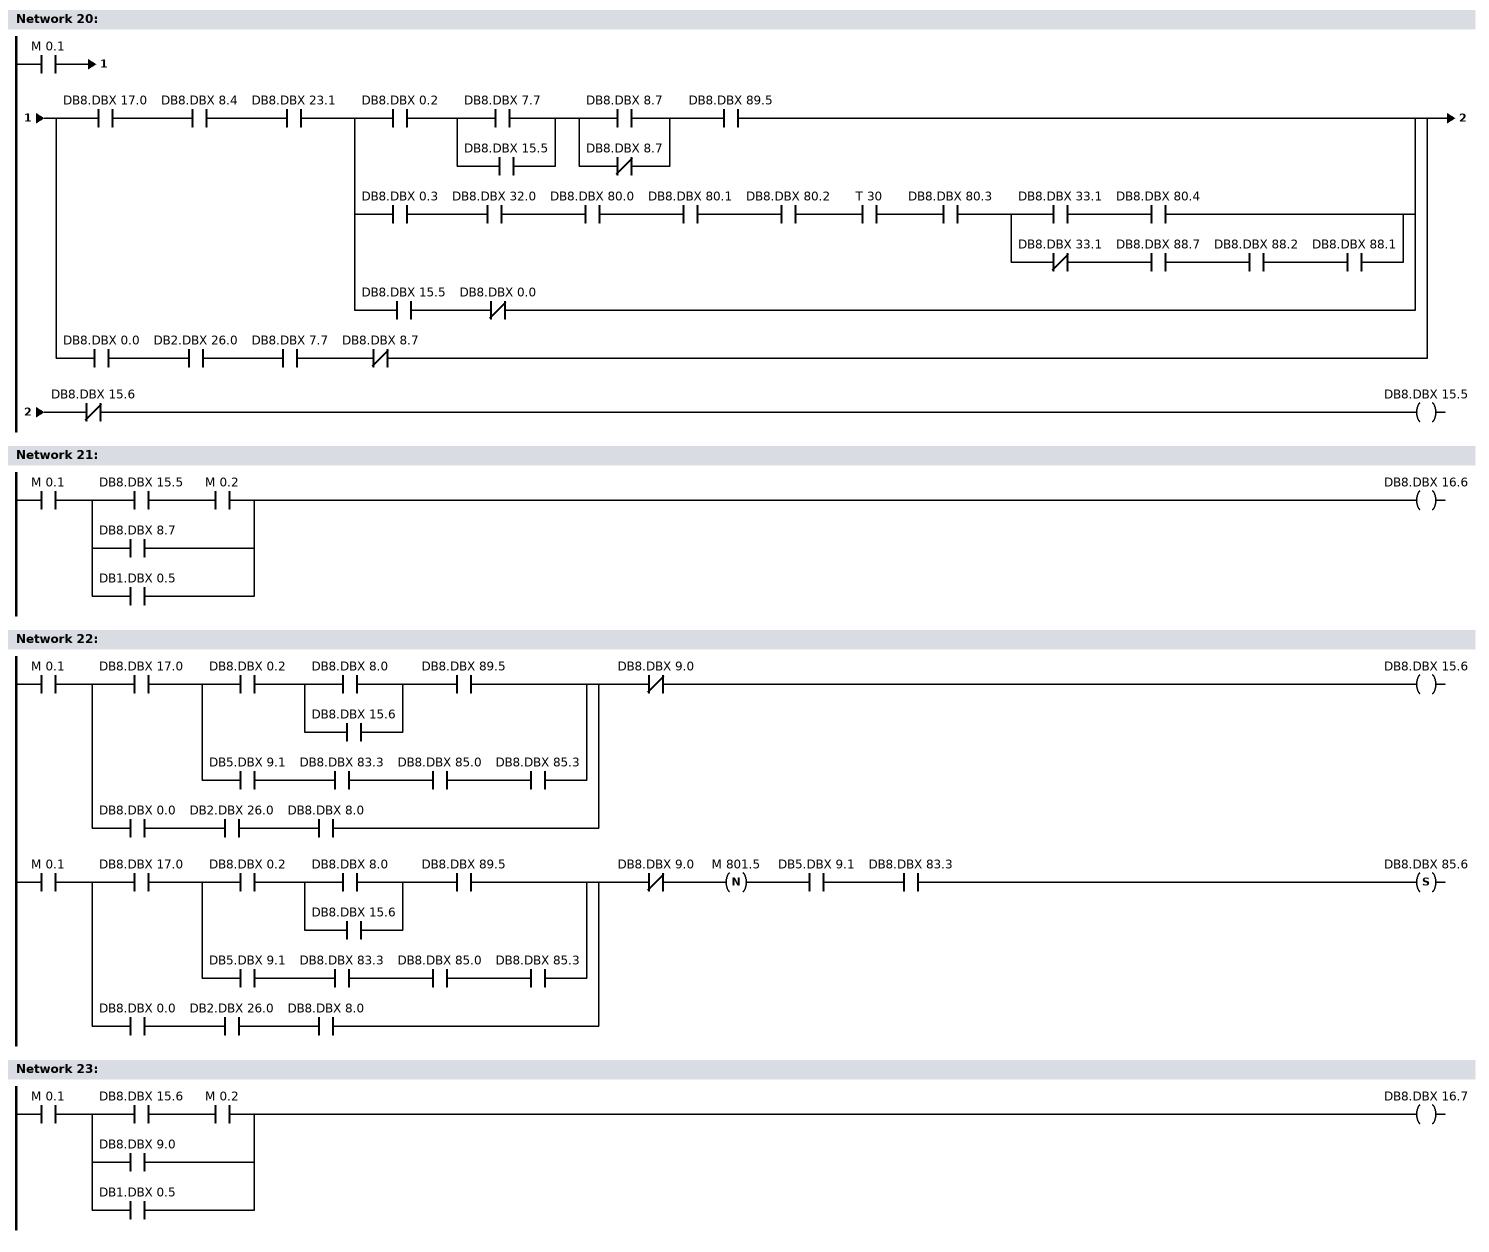
NETWORK
TITLE =
      A     M 0.1;
      A(;
      A     DB8.DBX 17.0;
      A     DB8.DBX 8.4;
      A     DB8.DBX 23.1;
      A(;
      A     DB8.DBX 0.2;
      A(;
      O     DB8.DBX 7.7;
      O     DB8.DBX 15.5;
      );
      A(;
      O     DB8.DBX 8.7;
      ON    DB8.DBX 8.7;
      );
      A     DB8.DBX 89.5;
      O;
      A     DB8.DBX 0.3;
      A     DB8.DBX 32.0;
      A     DB8.DBX 80.0;
      A     DB8.DBX 80.1;
      A     DB8.DBX 80.2;
      A     T 30;
      A     DB8.DBX 80.3;
      A(;
      A     DB8.DBX 33.1;
      A     DB8.DBX 80.4;
      O;
      AN    DB8.DBX 33.1;
      A     DB8.DBX 88.7;
      A     DB8.DBX 88.2;
      A     DB8.DBX 88.1;
      );
      O;
      A     DB8.DBX 15.5;
      AN    DB8.DBX 0.0;
      );
      O;
      A     DB8.DBX 0.0;
      A     DB2.DBX 26.0;
      A     DB8.DBX 7.7;
      AN    DB8.DBX 8.7;
      );
      AN    DB8.DBX 15.6;
      =     DB8.DBX 15.5;
NETWORK
TITLE =
      A     M 0.1;
      A(;
      A     DB8.DBX 15.5;
      A     M 0.2;
      O     DB8.DBX 8.7;
      O     DB1.DBX 0.5;
      );
      =     DB8.DBX 16.6;
NETWORK
TITLE =
      A     M 0.1;
      A(;
      A     DB8.DBX 17.0;
      A(;
      A     DB8.DBX 0.2;
      A(;
      O     DB8.DBX 8.0;
      O     DB8.DBX 15.6;
      );
      A     DB8.DBX 89.5;
      O;
      A     DB5.DBX 9.1;
      A     DB8.DBX 83.3;
      A     DB8.DBX 85.0;
      A     DB8.DBX 85.3;
      );
      O;
      A     DB8.DBX 0.0;
      A     DB2.DBX 26.0;
      A     DB8.DBX 8.0;
      );
      AN    DB8.DBX 9.0;
      =     L 0.0;
      A     L 0.0;
      BLD   102;
      =     DB8.DBX 15.6;
      A(;
      A     L 0.0;
      FN    M 801.5;
      );
      A     DB5.DBX 9.1;
      A     DB8.DBX 83.3;
      S     DB8.DBX 85.6;
NETWORK
TITLE =
      A     M 0.1;
      A(;
      A     DB8.DBX 15.6;
      A     M 0.2;
      O     DB8.DBX 9.0;
      O     DB1.DBX 0.5;
      );
      =     DB8.DBX 16.7;
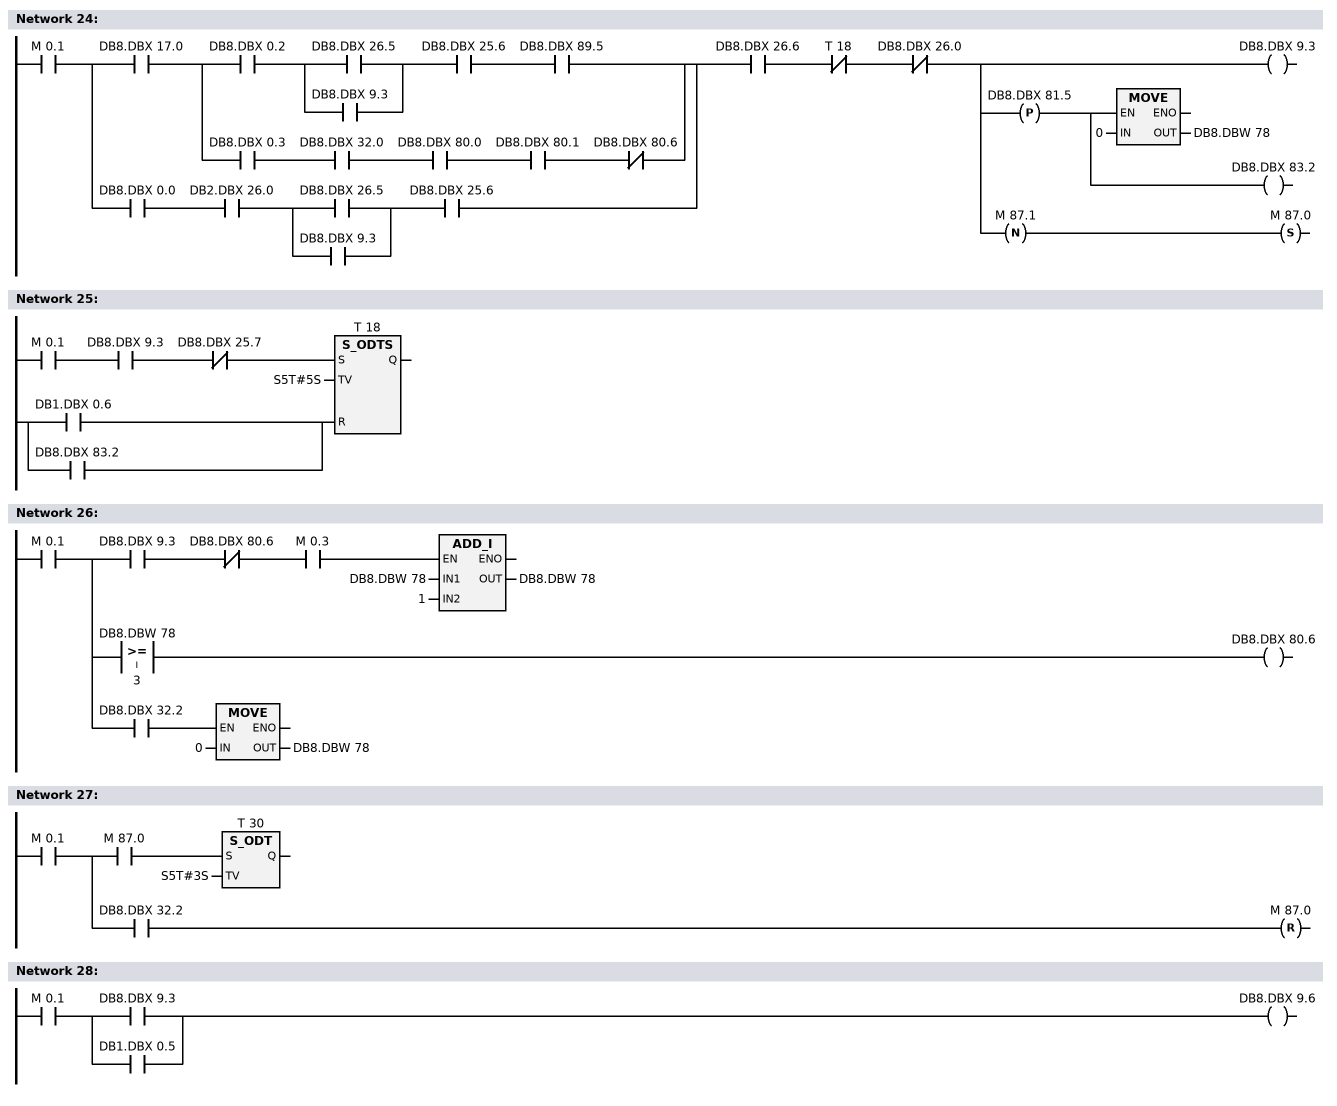
NETWORK
TITLE =
      A     M 0.1;
      A(;
      A     DB8.DBX 17.0;
      A(;
      A     DB8.DBX 0.2;
      A(;
      O     DB8.DBX 26.5;
      O     DB8.DBX 9.3;
      );
      A     DB8.DBX 25.6;
      A     DB8.DBX 89.5;
      O;
      A     DB8.DBX 0.3;
      A     DB8.DBX 32.0;
      A     DB8.DBX 80.0;
      A     DB8.DBX 80.1;
      AN    DB8.DBX 80.6;
      );
      O;
      A     DB8.DBX 0.0;
      A     DB2.DBX 26.0;
      A(;
      O     DB8.DBX 26.5;
      O     DB8.DBX 9.3;
      );
      A     DB8.DBX 25.6;
      );
      A     DB8.DBX 26.6;
      AN    T 18;
      AN    DB8.DBX 26.0;
      =     L 0.0;
      A     L 0.0;
      BLD   102;
      =     DB8.DBX 9.3;
      A     L 0.0;
      FP    DB8.DBX 81.5;
      =     L 0.1;
      A     L 0.1;
      JNB   M012;
      L     0;
      T     DB8.DBW 78;
M012: NOP   0;
      A     L 0.1;
      BLD   102;
      =     DB8.DBX 83.2;
      A     L 0.0;
      FN    M 87.1;
      S     M 87.0;
NETWORK
TITLE =
      A     M 0.1;
      A     DB8.DBX 9.3;
      AN    DB8.DBX 25.7;
      L     S5T#5S;
      SS    T 18;
      A(;
      O     DB1.DBX 0.6;
      O     DB8.DBX 83.2;
      );
      R     T 18;
      NOP   0;
      NOP   0;
      NOP   0;
NETWORK
TITLE =
      A     M 0.1;
      =     L 0.0;
      A     L 0.0;
      A     DB8.DBX 9.3;
      AN    DB8.DBX 80.6;
      A     M 0.3;
      JNB   M013;
      L     DB8.DBW 78;
      L     1;
      +I;
      T     DB8.DBW 78;
M013: NOP   0;
      A     L 0.0;
      A(;
      L     DB8.DBW 78;
      L     3;
      >=I;
      );
      =     DB8.DBX 80.6;
      A     L 0.0;
      A     DB8.DBX 32.2;
      JNB   M014;
      L     0;
      T     DB8.DBW 78;
M014: NOP   0;
NETWORK
TITLE =
      A     M 0.1;
      =     L 0.0;
      A     L 0.0;
      A     M 87.0;
      L     S5T#3S;
      SD    T 30;
      NOP   0;
      NOP   0;
      NOP   0;
      NOP   0;
      A     L 0.0;
      A     DB8.DBX 32.2;
      R     M 87.0;
NETWORK
TITLE =
      A     M 0.1;
      A(;
      O     DB8.DBX 9.3;
      O     DB1.DBX 0.5;
      );
      =     DB8.DBX 9.6;
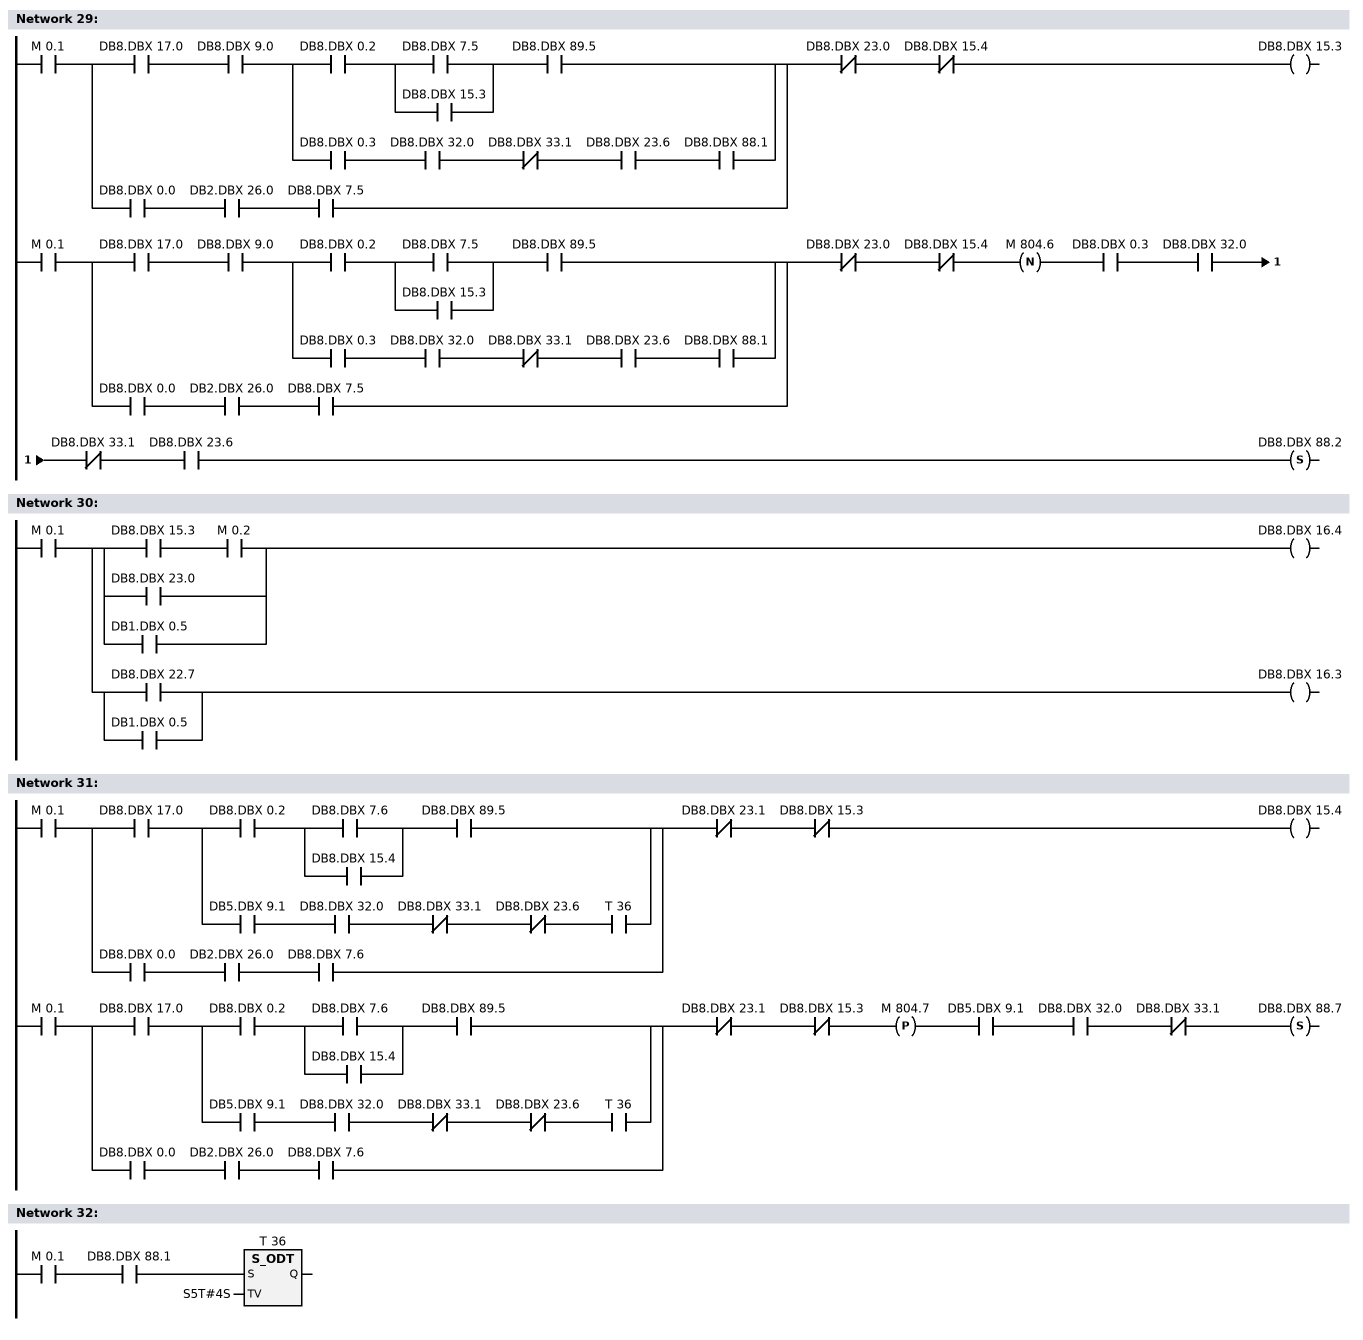
NETWORK
TITLE =
      A     M 0.1;
      A(;
      A     DB8.DBX 17.0;
      A     DB8.DBX 9.0;
      A(;
      A     DB8.DBX 0.2;
      A(;
      O     DB8.DBX 7.5;
      O     DB8.DBX 15.3;
      );
      A     DB8.DBX 89.5;
      O;
      A     DB8.DBX 0.3;
      A     DB8.DBX 32.0;
      AN    DB8.DBX 33.1;
      A     DB8.DBX 23.6;
      A     DB8.DBX 88.1;
      );
      O;
      A     DB8.DBX 0.0;
      A     DB2.DBX 26.0;
      A     DB8.DBX 7.5;
      );
      AN    DB8.DBX 23.0;
      AN    DB8.DBX 15.4;
      =     L 0.0;
      A     L 0.0;
      BLD   102;
      =     DB8.DBX 15.3;
      A(;
      A     L 0.0;
      FN    M 804.6;
      );
      A     DB8.DBX 0.3;
      A     DB8.DBX 32.0;
      AN    DB8.DBX 33.1;
      A     DB8.DBX 23.6;
      S     DB8.DBX 88.2;
NETWORK
TITLE =
      A     M 0.1;
      =     L 0.0;
      A     L 0.0;
      A(;
      A     DB8.DBX 15.3;
      A     M 0.2;
      O     DB8.DBX 23.0;
      O     DB1.DBX 0.5;
      );
      =     DB8.DBX 16.4;
      A     L 0.0;
      A(;
      O     DB8.DBX 22.7;
      O     DB1.DBX 0.5;
      );
      =     DB8.DBX 16.3;
NETWORK
TITLE =
      A     M 0.1;
      A(;
      A     DB8.DBX 17.0;
      A(;
      A     DB8.DBX 0.2;
      A(;
      O     DB8.DBX 7.6;
      O     DB8.DBX 15.4;
      );
      A     DB8.DBX 89.5;
      O;
      A     DB5.DBX 9.1;
      A     DB8.DBX 32.0;
      AN    DB8.DBX 33.1;
      AN    DB8.DBX 23.6;
      A     T 36;
      );
      O;
      A     DB8.DBX 0.0;
      A     DB2.DBX 26.0;
      A     DB8.DBX 7.6;
      );
      AN    DB8.DBX 23.1;
      AN    DB8.DBX 15.3;
      =     L 0.0;
      A     L 0.0;
      BLD   102;
      =     DB8.DBX 15.4;
      A(;
      A     L 0.0;
      FP    M 804.7;
      );
      A     DB5.DBX 9.1;
      A     DB8.DBX 32.0;
      AN    DB8.DBX 33.1;
      S     DB8.DBX 88.7;
NETWORK
TITLE =
      A     M 0.1;
      A     DB8.DBX 88.1;
      L     S5T#4S;
      SD    T 36;
      NOP   0;
      NOP   0;
      NOP   0;
      NOP   0;
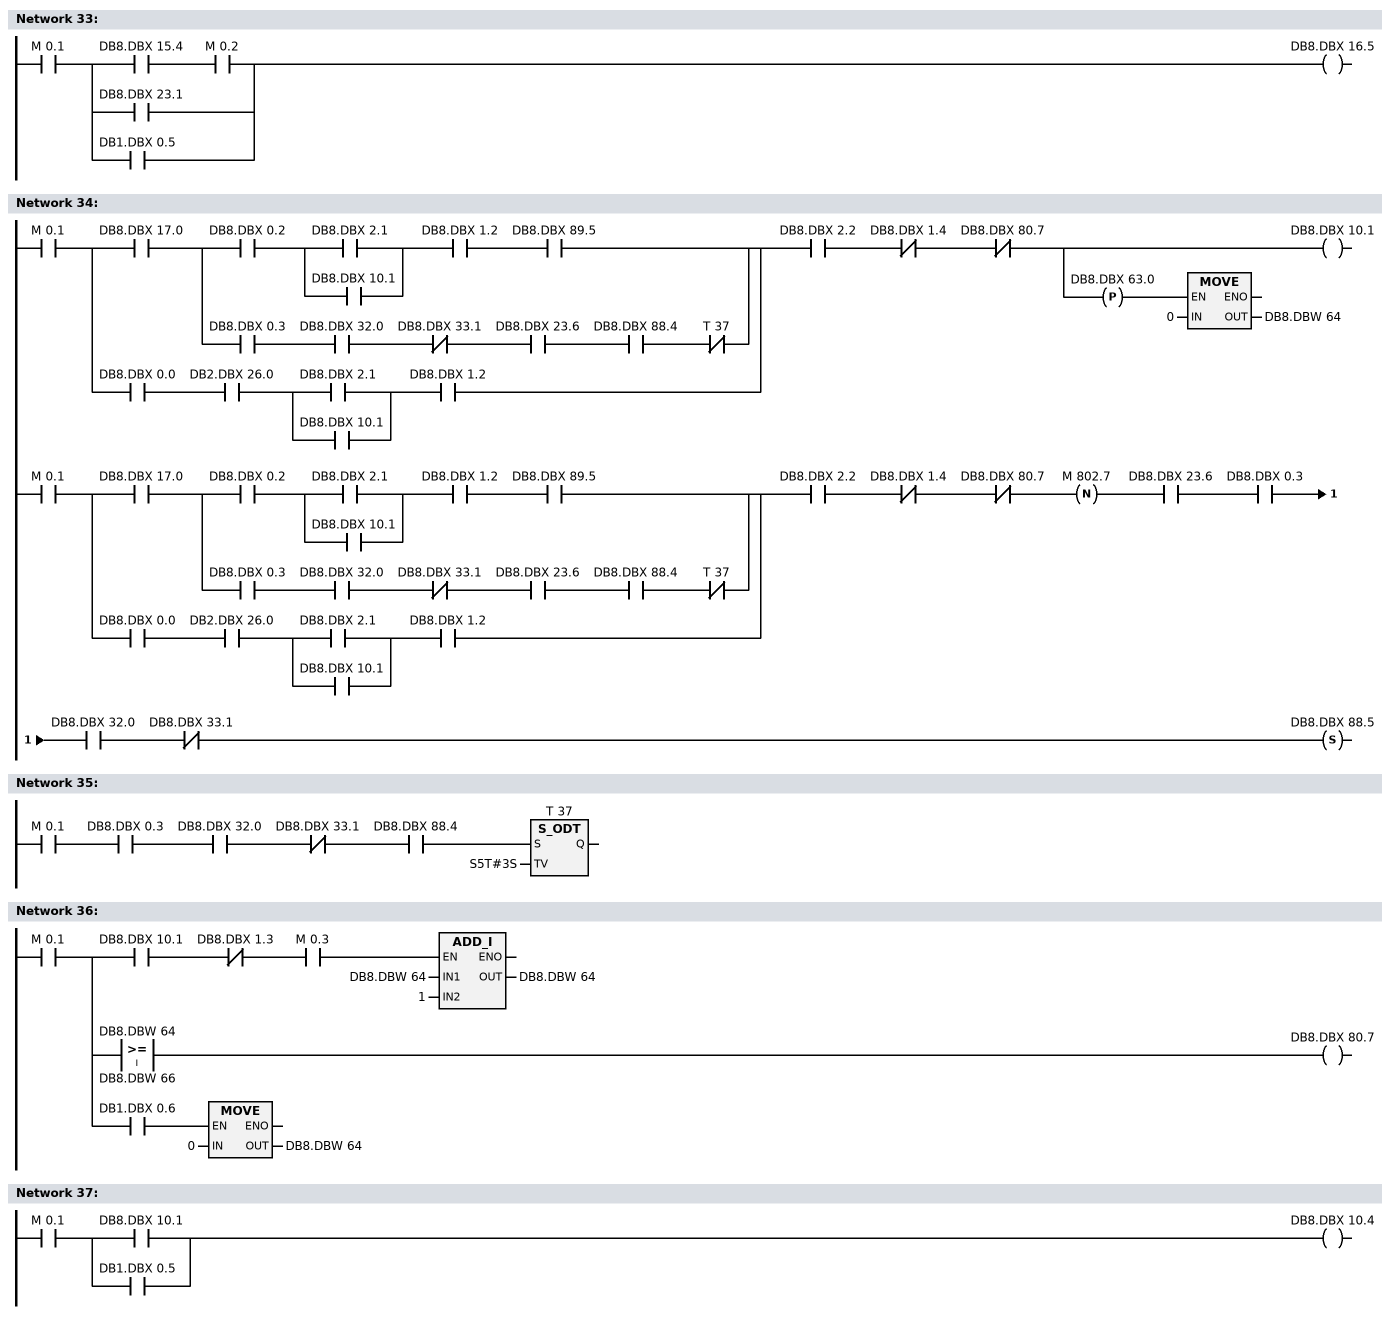
NETWORK
TITLE =
      A     M 0.1;
      A(;
      A     DB8.DBX 15.4;
      A     M 0.2;
      O     DB8.DBX 23.1;
      O     DB1.DBX 0.5;
      );
      =     DB8.DBX 16.5;
NETWORK
TITLE =
      A     M 0.1;
      A(;
      A     DB8.DBX 17.0;
      A(;
      A     DB8.DBX 0.2;
      A(;
      O     DB8.DBX 2.1;
      O     DB8.DBX 10.1;
      );
      A     DB8.DBX 1.2;
      A     DB8.DBX 89.5;
      O;
      A     DB8.DBX 0.3;
      A     DB8.DBX 32.0;
      AN    DB8.DBX 33.1;
      A     DB8.DBX 23.6;
      A     DB8.DBX 88.4;
      AN    T 37;
      );
      O;
      A     DB8.DBX 0.0;
      A     DB2.DBX 26.0;
      A(;
      O     DB8.DBX 2.1;
      O     DB8.DBX 10.1;
      );
      A     DB8.DBX 1.2;
      );
      A     DB8.DBX 2.2;
      AN    DB8.DBX 1.4;
      AN    DB8.DBX 80.7;
      =     L 0.0;
      A     L 0.0;
      BLD   102;
      =     DB8.DBX 10.1;
      A     L 0.0;
      FP    DB8.DBX 63.0;
      JNB   M015;
      L     0;
      T     DB8.DBW 64;
M015: NOP   0;
      A(;
      A     L 0.0;
      FN    M 802.7;
      );
      A     DB8.DBX 23.6;
      A     DB8.DBX 0.3;
      A     DB8.DBX 32.0;
      AN    DB8.DBX 33.1;
      S     DB8.DBX 88.5;
NETWORK
TITLE =
      A     M 0.1;
      A     DB8.DBX 0.3;
      A     DB8.DBX 32.0;
      AN    DB8.DBX 33.1;
      A     DB8.DBX 88.4;
      L     S5T#3S;
      SD    T 37;
      NOP   0;
      NOP   0;
      NOP   0;
      NOP   0;
NETWORK
TITLE =
      A     M 0.1;
      =     L 0.0;
      A     L 0.0;
      A     DB8.DBX 10.1;
      AN    DB8.DBX 1.3;
      A     M 0.3;
      JNB   M016;
      L     DB8.DBW 64;
      L     1;
      +I;
      T     DB8.DBW 64;
M016: NOP   0;
      A     L 0.0;
      A(;
      L     DB8.DBW 64;
      L     DB8.DBW 66;
      >=I;
      );
      =     DB8.DBX 80.7;
      A     L 0.0;
      A     DB1.DBX 0.6;
      JNB   M017;
      L     0;
      T     DB8.DBW 64;
M017: NOP   0;
NETWORK
TITLE =
      A     M 0.1;
      A(;
      O     DB8.DBX 10.1;
      O     DB1.DBX 0.5;
      );
      =     DB8.DBX 10.4;
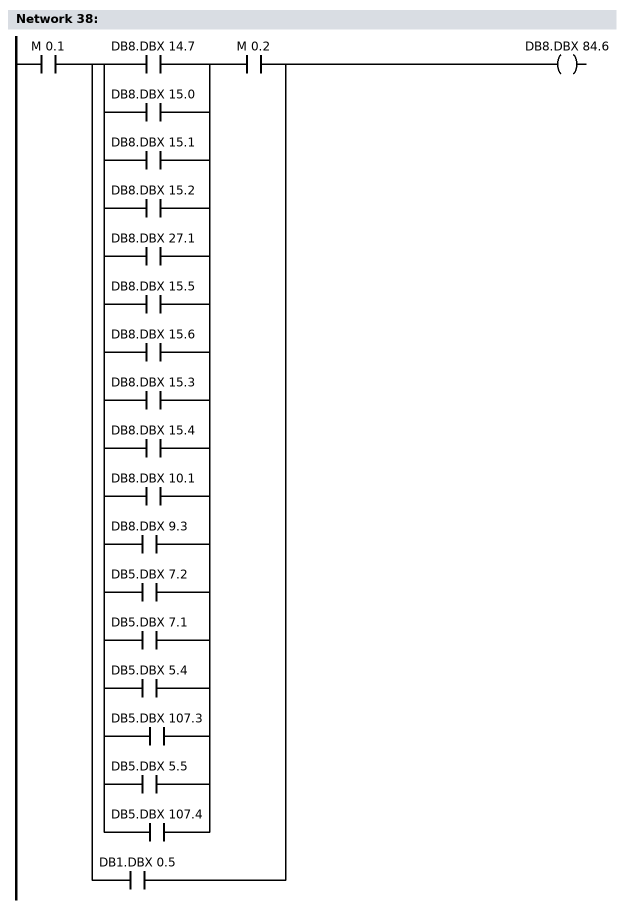
NETWORK
TITLE =
      A     M 0.1;
      A(;
      A(;
      O     DB8.DBX 14.7;
      O     DB8.DBX 15.0;
      O     DB8.DBX 15.1;
      O     DB8.DBX 15.2;
      O     DB8.DBX 27.1;
      O     DB8.DBX 15.5;
      O     DB8.DBX 15.6;
      O     DB8.DBX 15.3;
      O     DB8.DBX 15.4;
      O     DB8.DBX 10.1;
      O     DB8.DBX 9.3;
      O     DB5.DBX 7.2;
      O     DB5.DBX 7.1;
      O     DB5.DBX 5.4;
      O     DB5.DBX 107.3;
      O     DB5.DBX 5.5;
      O     DB5.DBX 107.4;
      );
      A     M 0.2;
      O     DB1.DBX 0.5;
      );
      =     DB8.DBX 84.6;
END_FUNCTION

FUNCTION FC 21 : VOID
AUTHOR : Arun
VERSION : 0.1
BEGIN
// (block stored without names or comments; labels and parameter names are numbered)
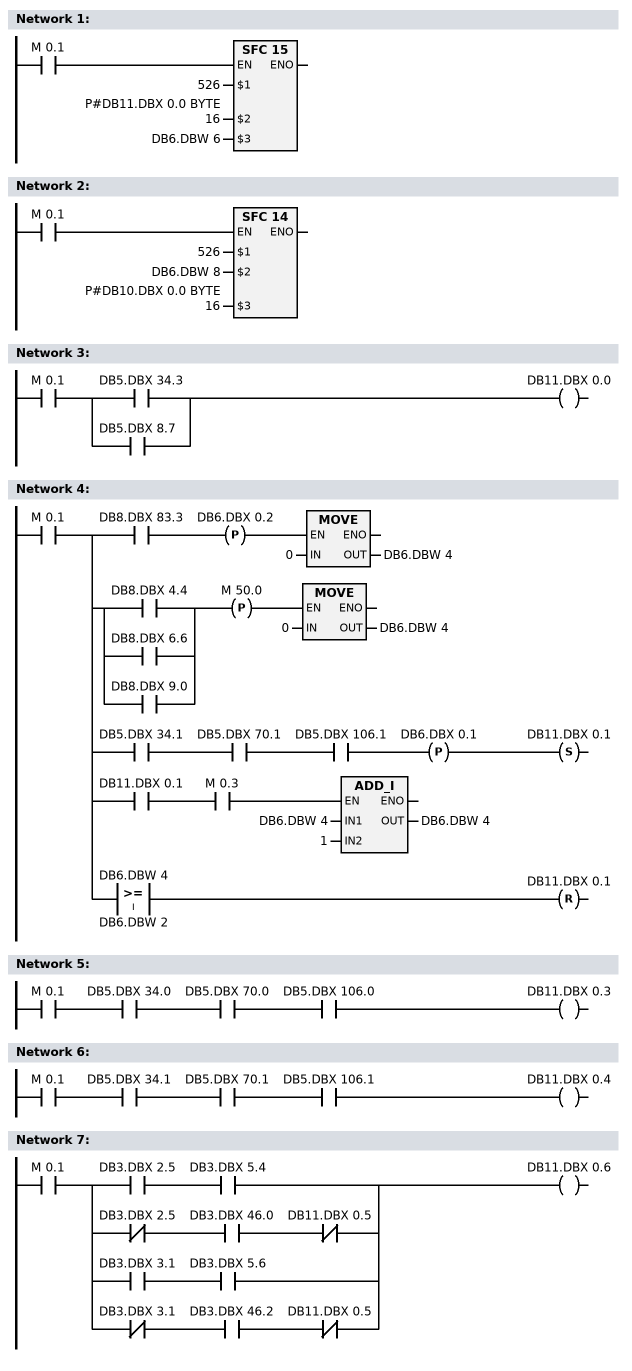
NETWORK
TITLE =
      A     M 0.1;
      JNB   M001;
      CALL  SFC 15 (
           $1                       := 526,
           $2                       := P#DB11.DBX 0.0 BYTE 16,
           $3                       := DB6.DBW 6);
M001: NOP   0;
NETWORK
TITLE =
      A     M 0.1;
      JNB   M002;
      CALL  SFC 14 (
           $1                       := 526,
           $2                       := DB6.DBW 8,
           $3                       := P#DB10.DBX 0.0 BYTE 16);
M002: NOP   0;
NETWORK
TITLE =
      A     M 0.1;
      A(;
      O     DB5.DBX 34.3;
      O     DB5.DBX 8.7;
      );
      =     DB11.DBX 0.0;
NETWORK
TITLE =
      A     M 0.1;
      =     L 0.0;
      A     L 0.0;
      A     DB8.DBX 83.3;
      FP    DB6.DBX 0.2;
      JNB   M003;
      L     0;
      T     DB6.DBW 4;
M003: NOP   0;
      A     L 0.0;
      A(;
      O     DB8.DBX 4.4;
      O     DB8.DBX 6.6;
      O     DB8.DBX 9.0;
      );
      FP    M 50.0;
      JNB   M004;
      L     0;
      T     DB6.DBW 4;
M004: NOP   0;
      A     L 0.0;
      A     DB5.DBX 34.1;
      A     DB5.DBX 70.1;
      A     DB5.DBX 106.1;
      FP    DB6.DBX 0.1;
      S     DB11.DBX 0.1;
      A     L 0.0;
      A     DB11.DBX 0.1;
      A     M 0.3;
      JNB   M005;
      L     DB6.DBW 4;
      L     1;
      +I;
      T     DB6.DBW 4;
M005: NOP   0;
      A     L 0.0;
      A(;
      L     DB6.DBW 4;
      L     DB6.DBW 2;
      >=I;
      );
      R     DB11.DBX 0.1;
NETWORK
TITLE =
      A     M 0.1;
      A     DB5.DBX 34.0;
      A     DB5.DBX 70.0;
      A     DB5.DBX 106.0;
      =     DB11.DBX 0.3;
NETWORK
TITLE =
      A     M 0.1;
      A     DB5.DBX 34.1;
      A     DB5.DBX 70.1;
      A     DB5.DBX 106.1;
      =     DB11.DBX 0.4;
NETWORK
TITLE =
      A     M 0.1;
      A(;
      A     DB3.DBX 2.5;
      A     DB3.DBX 5.4;
      O;
      AN    DB3.DBX 2.5;
      A     DB3.DBX 46.0;
      AN    DB11.DBX 0.5;
      O;
      A     DB3.DBX 3.1;
      A     DB3.DBX 5.6;
      O;
      AN    DB3.DBX 3.1;
      A     DB3.DBX 46.2;
      AN    DB11.DBX 0.5;
      );
      =     DB11.DBX 0.6;
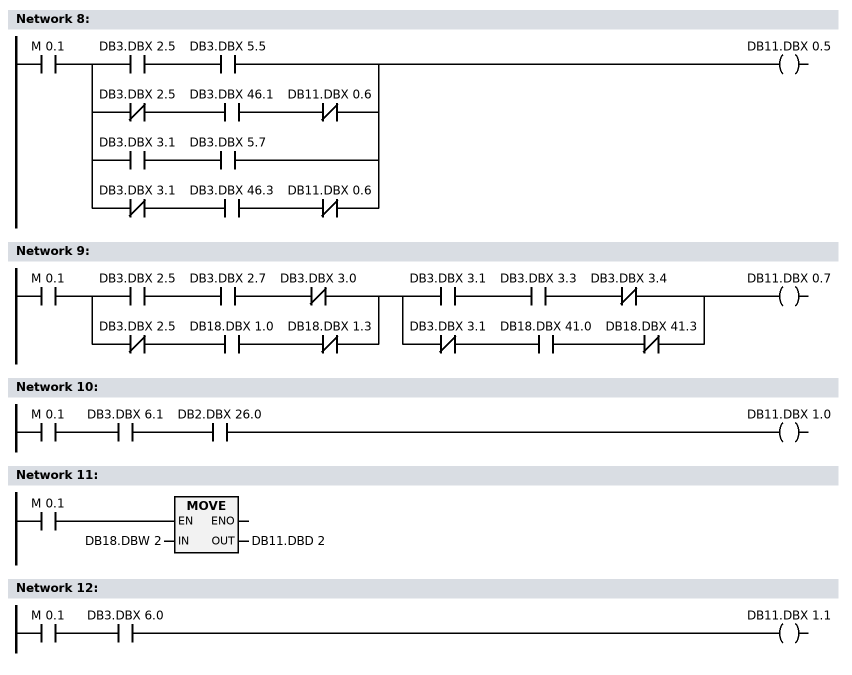
NETWORK
TITLE =
      A     M 0.1;
      A(;
      A     DB3.DBX 2.5;
      A     DB3.DBX 5.5;
      O;
      AN    DB3.DBX 2.5;
      A     DB3.DBX 46.1;
      AN    DB11.DBX 0.6;
      O;
      A     DB3.DBX 3.1;
      A     DB3.DBX 5.7;
      O;
      AN    DB3.DBX 3.1;
      A     DB3.DBX 46.3;
      AN    DB11.DBX 0.6;
      );
      =     DB11.DBX 0.5;
NETWORK
TITLE =
      A     M 0.1;
      A(;
      A     DB3.DBX 2.5;
      A     DB3.DBX 2.7;
      AN    DB3.DBX 3.0;
      O;
      AN    DB3.DBX 2.5;
      A     DB18.DBX 1.0;
      AN    DB18.DBX 1.3;
      );
      A(;
      A     DB3.DBX 3.1;
      A     DB3.DBX 3.3;
      AN    DB3.DBX 3.4;
      O;
      AN    DB3.DBX 3.1;
      A     DB18.DBX 41.0;
      AN    DB18.DBX 41.3;
      );
      =     DB11.DBX 0.7;
NETWORK
TITLE =
      A     M 0.1;
      A     DB3.DBX 6.1;
      A     DB2.DBX 26.0;
      =     DB11.DBX 1.0;
NETWORK
TITLE =
      A     M 0.1;
      JNB   M006;
      L     DB18.DBW 2;
      T     DB11.DBD 2;
M006: NOP   0;
NETWORK
TITLE =
      A     M 0.1;
      A     DB3.DBX 6.0;
      =     DB11.DBX 1.1;
END_FUNCTION

// FC 105: know-how protected block, not included

// FC 106: know-how protected block, not included

DATA_BLOCK DB 1
VERSION : 0.1
BEGIN
// 12 bytes; values not shown
END_DATA_BLOCK

DATA_BLOCK DB 2
VERSION : 0.1
BEGIN
// 38 bytes; values not shown
END_DATA_BLOCK

DATA_BLOCK DB 3
VERSION : 0.1
BEGIN
// 60 bytes; values not shown
END_DATA_BLOCK

DATA_BLOCK DB 4
VERSION : 0.1
BEGIN
// 20 bytes; values not shown
END_DATA_BLOCK

DATA_BLOCK DB 5
VERSION : 0.1
BEGIN
// 120 bytes; values not shown
END_DATA_BLOCK

DATA_BLOCK DB 6
VERSION : 0.1
BEGIN
// 10 bytes; values not shown
END_DATA_BLOCK

DATA_BLOCK DB 7
VERSION : 0.1
UDT 2
BEGIN
END_DATA_BLOCK

DATA_BLOCK DB 8
VERSION : 0.1
BEGIN
// 90 bytes; values not shown
END_DATA_BLOCK

DATA_BLOCK DB 10
VERSION : 0.1
BEGIN
// 18 bytes; values not shown
END_DATA_BLOCK

DATA_BLOCK DB 11
VERSION : 0.1
BEGIN
// 18 bytes; values not shown
END_DATA_BLOCK

DATA_BLOCK DB 15
VERSION : 0.1
BEGIN
// 44 bytes; values not shown
END_DATA_BLOCK

DATA_BLOCK DB 17
VERSION : 0.1
BEGIN
// 24 bytes; values not shown
END_DATA_BLOCK

DATA_BLOCK DB 18
VERSION : 0.1
BEGIN
// 80 bytes; values not shown
END_DATA_BLOCK

DATA_BLOCK DB 19
VERSION : 0.1
BEGIN
// 120 bytes; values not shown
END_DATA_BLOCK

ORGANIZATION_BLOCK OB 1
AUTHOR : Arun_Ram
VERSION : 0.1
BEGIN
// (block stored without names or comments; labels and parameter names are numbered)
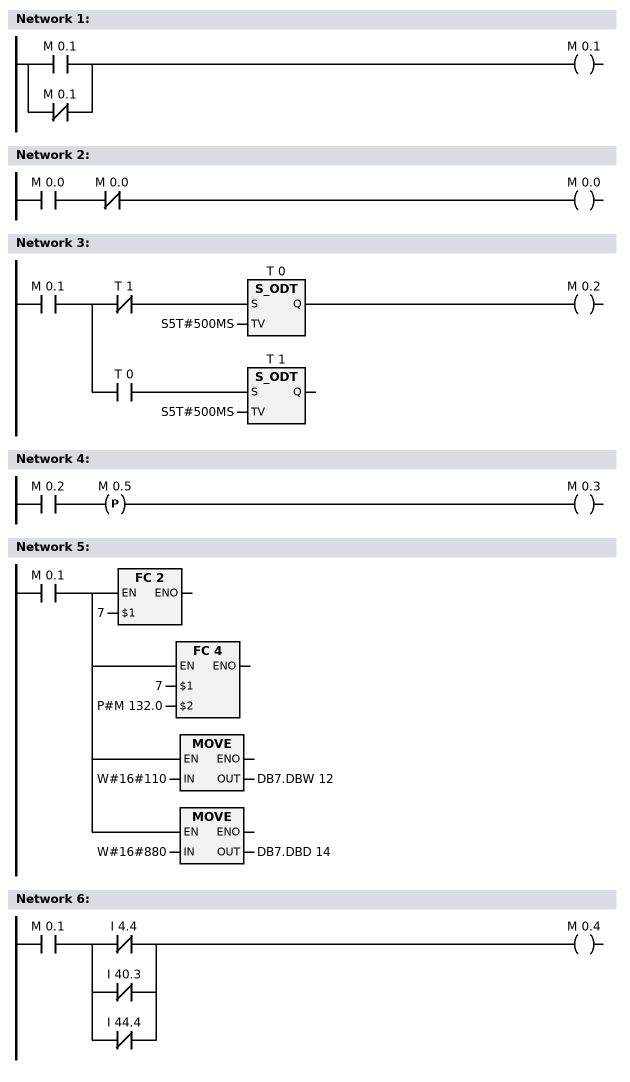
NETWORK
TITLE =
      O     M 0.1;
      ON    M 0.1;
      =     M 0.1;
NETWORK
TITLE =
      A     M 0.0;
      AN    M 0.0;
      =     M 0.0;
NETWORK
TITLE =
      A     M 0.1;
      =     L 22.0;
      A     L 22.0;
      AN    T 1;
      L     S5T#500MS;
      SD    T 0;
      NOP   0;
      NOP   0;
      NOP   0;
      A     T 0;
      =     M 0.2;
      A     L 22.0;
      A     T 0;
      L     S5T#500MS;
      SD    T 1;
      NOP   0;
      NOP   0;
      NOP   0;
      NOP   0;
NETWORK
TITLE =
      A     M 0.2;
      FP    M 0.5;
      =     M 0.3;
NETWORK
TITLE =
      A     M 0.1;
      =     L 22.0;
      A     L 22.0;
      JNB   M001;
      CALL  FC 2 (
           $1                       := 7);
M001: NOP   0;
      A     L 22.0;
      JNB   M002;
      CALL  FC 4 (
           $1                       := 7,
           $2                       := P#M 132.0);
M002: NOP   0;
      A     L 22.0;
      JNB   M003;
      L     W#16#110;
      T     DB7.DBW 12;
M003: NOP   0;
      A     L 22.0;
      JNB   M004;
      L     W#16#880;
      T     DB7.DBD 14;
M004: NOP   0;
NETWORK
TITLE =
      A     M 0.1;
      A(;
      ON    I 4.4;
      ON    I 40.3;
      ON    I 44.4;
      );
      =     M 0.4;
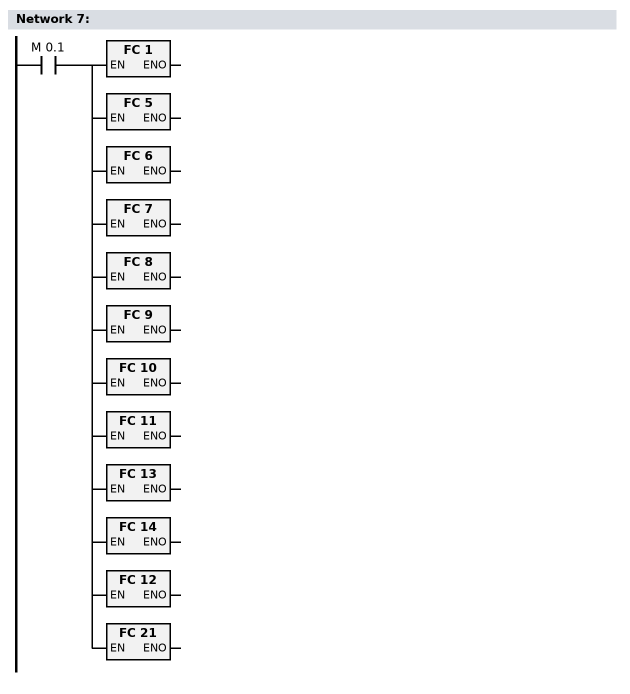
NETWORK
TITLE =
      A     M 0.1;
      =     L 22.0;
      A     L 22.0;
      JNB   M005;
      CALL  FC 1;
M005: NOP   0;
      A     L 22.0;
      JNB   M006;
      CALL  FC 5;
M006: NOP   0;
      A     L 22.0;
      JNB   M007;
      CALL  FC 6;
M007: NOP   0;
      A     L 22.0;
      JNB   M008;
      CALL  FC 7;
M008: NOP   0;
      A     L 22.0;
      JNB   M009;
      CALL  FC 8;
M009: NOP   0;
      A     L 22.0;
      JNB   M010;
      CALL  FC 9;
M010: NOP   0;
      A     L 22.0;
      JNB   M011;
      CALL  FC 10;
M011: NOP   0;
      A     L 22.0;
      JNB   M012;
      CALL  FC 11;
M012: NOP   0;
      A     L 22.0;
      JNB   M013;
      CALL  FC 13;
M013: NOP   0;
      A     L 22.0;
      JNB   M014;
      CALL  FC 14;
M014: NOP   0;
      A     L 22.0;
      JNB   M015;
      CALL  FC 12;
M015: NOP   0;
      A     L 22.0;
      JNB   M016;
      CALL  FC 21;
M016: NOP   0;
END_ORGANIZATION_BLOCK

ORGANIZATION_BLOCK OB 80
VERSION : 0.1
BEGIN
// (block stored without names or comments; labels and parameter names are numbered)
END_ORGANIZATION_BLOCK

ORGANIZATION_BLOCK OB 82
VERSION : 0.1
BEGIN
// (block stored without names or comments; labels and parameter names are numbered)
END_ORGANIZATION_BLOCK

ORGANIZATION_BLOCK OB 85
VERSION : 0.1
BEGIN
// (block stored without names or comments; labels and parameter names are numbered)
END_ORGANIZATION_BLOCK

ORGANIZATION_BLOCK OB 86
VERSION : 0.1
BEGIN
// (block stored without names or comments; labels and parameter names are numbered)
END_ORGANIZATION_BLOCK

ORGANIZATION_BLOCK OB 87
VERSION : 0.1
BEGIN
// (block stored without names or comments; labels and parameter names are numbered)
END_ORGANIZATION_BLOCK

ORGANIZATION_BLOCK OB 100
VERSION : 0.1
BEGIN
// (block stored without names or comments; labels and parameter names are numbered)
NETWORK
TITLE =
END_ORGANIZATION_BLOCK

ORGANIZATION_BLOCK OB 121
VERSION : 0.1
BEGIN
// (block stored without names or comments; labels and parameter names are numbered)
END_ORGANIZATION_BLOCK

ORGANIZATION_BLOCK OB 122
VERSION : 0.1
BEGIN
// (block stored without names or comments; labels and parameter names are numbered)
END_ORGANIZATION_BLOCK
